	// === OPERATOR INTERFACE VALIDATION ===
	// Verify flags provide clear indication to operators
	IF eTestResult = E_CommandResult.Ok THEN
		AssertTrue(
			Condition := (iTestCommand.P_CommandStatus.BaseStatus.Done = TRUE) AND
						 (iTestCommand.P_CommandStatus.BaseStatus.Busy = FALSE) AND
						 (iTestCommand.P_CommandStatus.BaseStatus.Error = FALSE),
			Message := CONCAT(sTestScenario, ': OPERATOR - Success indication: Done=TRUE + Busy=FALSE + Error=FALSE')
		);
	ELSE
		AssertTrue(
			Condition := (iTestCommand.P_CommandStatus.BaseStatus.Error = TRUE) AND
						 (iTestCommand.P_CommandStatus.BaseStatus.Busy = FALSE),
			Message := CONCAT(sTestScenario, ': OPERATOR - Error indication: Error=TRUE + Busy=FALSE')
		);
	END_IF

	// Reset for next iteration
	iTestCommand.Reset();
END_FOR

TEST_FINISHED();
END_METHOD

METHOD PRIVATE TEST_Config_FallbackToLocal_WhenInjectedInvalid
VAR
	TestIdx : DINT := INDEX_CONFIG_FALLBACKTOLOCAL_WHENINJECTEDINVALID;
    configResolution : E_ConfigurationResolution;
END_VAR
TEST(__POUNAME());

// Purpose: Verify command falls back to local configuration when injected interfaces become invalid
// Tests resilient configuration resolution

// Initialize test objects - Use index 204 to avoid conflicts
TestCommand[TestIdx].Initialize();
TestComponent[TestIdx].Initialize();
TestCommandConfig[TestIdx].Initialize();
TestPermIntlk[TestIdx].Initialize();

// Safe interface assignments using __QUERYINTERFACE for validation
iTestCommand := TestCommand[TestIdx];

iTestCommandConfig := TestCommandConfig[TestIdx];

iTestComponent := TestComponent[TestIdx];

iTestPermIntlkConfig := TestPermIntlk[TestIdx];

// Interface validation
IF iTestCommand = 0 THEN
    AssertTrue(Condition := FALSE, Message := 'TEST FAILED: iTestCommand interface is null');
    RETURN;
END_IF

// === STEP 1: Initially Use Local Configuration ===
// Don't inject configurations - should use local fallback
TestCommand[TestIdx].Initialize();

// Verify local configuration is being used
configResolution := TestCommand[TestIdx].P_CommandStatus.CmdConfigurationResolution;
AssertEquals_INT(
    Expected := E_ConfigurationResolution.Local,
    Actual := configResolution,
    Message := 'Should use Local configuration when no interfaces injected'
);

// === STEP 2: Inject Valid Configurations ===
// Configure valid injected configuration
TestCommandConfig[TestIdx].P_CommandConfiguration.CommandDescription := 'Injected Valid Config';
TestCommandConfig[TestIdx].P_CommandConfiguration.TimeoutTime := T#15S;
TestCommandConfig[TestIdx].P_CommandConfiguration.RetryCountONLYFORCOMMSENDS := 5;

// Configure permissive to be OK for successful validation and execution
IF iTestPermIntlkConfig <> 0 THEN
	iTestPermIntlkConfig.P_PermIntlkConfiguration.PermIntlkObj[1].Description := 'Fallback Test Permissive';
	iTestPermIntlkConfig.P_PermIntlkConfiguration.PermIntlkObj[1].Condition := TRUE;
	iTestPermIntlkConfig.P_PermIntlkConfiguration.PermIntlkObj[1].Index := 1;
	TestPermIntlk[TestIdx].CyclicLogic(); // Update permissive evaluation
END_IF

// Inject configurations
iTestCommand.InjectConfigurations(
    iComponent := iTestComponent,
    iCommandConfiguration := iTestCommandConfig,
    iPermIntlkConfiguration := iTestPermIntlkConfig
);

// Resolve configurations after injection
iTestCommand.CyclicLogic();

// Verify injected configuration is being used
configResolution := iTestCommand.P_CommandStatus.CmdConfigurationResolution;
AssertEquals_INT(
    Expected := E_ConfigurationResolution.InjectedInterface,
    Actual := configResolution,
    Message := 'Should use InjectedInterface configuration when valid interfaces provided'
);

// Verify we can access injected configuration
AssertEquals_STRING(
    Expected := 'Injected Valid Config',
    Actual := TestCommand[TestIdx].P_CommandStatus.ConfigRef.CommandDescription,
    Message := 'Should access injected configuration description'
);

AssertEquals_TIME(
    Expected := T#15S,
    Actual := TestCommand[TestIdx].P_CommandStatus.ConfigRef.TimeoutTime,
    Message := 'Should access injected configuration timeout'
);

// === STEP 3: Simulate Configuration Becoming Invalid ===
// This tests runtime resilience when external configuration becomes corrupted
// In real systems, this could happen due to network issues, memory corruption, etc.

// Inject null interfaces to simulate failure
iTestCommand.InjectConfigurations(
    iComponent := iTestComponent,
    iCommandConfiguration := 0, // Null interface
    iPermIntlkConfiguration := 0  // Null interface
);

// Re-initialize to trigger configuration resolution
TestCommand[TestIdx].Initialize();

// Trigger configuration resolution after invalidation
iTestCommand.CyclicLogic();

// === STEP 4: Verify Fallback to Local Configuration ===
configResolution := TestCommand[TestIdx].P_CommandStatus.CmdConfigurationResolution;
AssertEquals_INT(
    Expected := E_ConfigurationResolution.Local,
    Actual := configResolution,
    Message := 'RESILIENCE: Should fallback to Local configuration when injected becomes invalid'
);

// Verify local configuration is accessible and provides default values
AssertEquals_STRING(
    Expected := 'Missing Command Configuration Interface Reference',
    Actual := TestCommand[TestIdx].LocalCommandConfiguration.CommandDescription,
    Message := 'Should use local fallback configuration description'
);

// === STEP 5: Command Should Still Function with Local Configuration ===
// Even with fallback configuration, basic command operations should work
iTestCommand.Execute();

// Command should accept execution even with local configuration
AssertEquals_UDINT(
    Expected := E_CommandResult.Accepted,
    Actual := iTestCommand.P_CommandStatus.Result,
    Message := 'Command should function with local fallback configuration'
);

// Progress through states
iTestCommand.CyclicLogic(); // Idle → Execute
iTestCommand.CyclicLogic(); // Execute → Monitor
iTestCommand.Complete(); // Signal completion
iTestCommand.CyclicLogic(); // Monitor → Complete

// Should complete successfully
AssertEquals_UDINT(
    Expected := E_CommandState.Complete,
    Actual := iTestCommand.P_CommandStatus.StepState,
    Message := 'Command should complete successfully with local configuration'
);

AssertEquals_UDINT(
    Expected := E_CommandResult.Ok,
    Actual := iTestCommand.P_CommandStatus.Result,
    Message := 'Command should have Ok result with local configuration'
);

TEST_FINISHED();
END_METHOD

METHOD PRIVATE TEST_Config_RecoveryToInjected_WhenValidAgain
VAR
	TestIdx : DINT := INDEX_CONFIG_RECOVERYTOINJECTED_WHENVALIDAGAIN;
    configResolution : E_ConfigurationResolution;
END_VAR
TEST(__POUNAME());

// Purpose: Verify command can recover to injected configuration when it becomes valid again
// Tests configuration resolution recovery mechanism

// Initialize test objects - Use index 205 to avoid conflicts
TestCommand[TestIdx].Initialize();
TestComponent[TestIdx].Initialize();
TestCommandConfig[TestIdx].Initialize();
TestPermIntlk[TestIdx].Initialize();

// Safe interface assignments using __QUERYINTERFACE for validation
iTestCommand := TestCommand[TestIdx];

iTestCommandConfig := TestCommandConfig[TestIdx];

iTestComponent := TestComponent[TestIdx];

iTestPermIntlkConfig := TestPermIntlk[TestIdx];

// Interface validation
IF iTestCommand = 0 THEN
    AssertTrue(Condition := FALSE, Message := 'TEST FAILED: iTestCommand interface is null');
    RETURN;
END_IF

// === STEP 1: Start with Local Configuration ===
TestCommand[TestIdx].Initialize();

configResolution := TestCommand[TestIdx].P_CommandStatus.CmdConfigurationResolution;
AssertEquals_INT(
    Expected := E_ConfigurationResolution.Local,
    Actual := configResolution,
    Message := 'Should start with Local configuration'
);

// === STEP 2: Inject Invalid Configuration (Null Interfaces) ===
iTestCommand.InjectConfigurations(
    iComponent := iTestComponent,
    iCommandConfiguration := 0, // Null interface
    iPermIntlkConfiguration := 0  // Null interface
);

TestCommand[TestIdx].Initialize();

// Should still use local configuration
configResolution := TestCommand[TestIdx].P_CommandStatus.CmdConfigurationResolution;
AssertEquals_INT(
    Expected := E_ConfigurationResolution.Local,
    Actual := configResolution,
    Message := 'Should remain with Local configuration when invalid injected'
);

// === STEP 3: Inject Valid Configuration ===
// Configure a distinctive injected configuration for recovery test
TestCommandConfig[TestIdx].P_CommandConfiguration.CommandDescription := 'Recovered Injected Config';
TestCommandConfig[TestIdx].P_CommandConfiguration.TimeoutTime := T#25S;
TestCommandConfig[TestIdx].P_CommandConfiguration.RetryCountONLYFORCOMMSENDS := 7;

// Configure permissive to be OK for successful validation and execution
IF iTestPermIntlkConfig <> 0 THEN
	iTestPermIntlkConfig.P_PermIntlkConfiguration.PermIntlkObj[1].Description := 'Recovery Test Permissive';
	iTestPermIntlkConfig.P_PermIntlkConfiguration.PermIntlkObj[1].Condition := TRUE;
	iTestPermIntlkConfig.P_PermIntlkConfiguration.PermIntlkObj[1].Index := 1;
	TestPermIntlk[TestIdx].CyclicLogic(); // Update permissive evaluation
END_IF

// Inject valid configurations
iTestCommand.InjectConfigurations(
    iComponent := iTestComponent,
    iCommandConfiguration := iTestCommandConfig,
    iPermIntlkConfiguration := iTestPermIntlkConfig
);

// Resolve configurations after injection
iTestCommand.CyclicLogic();

// Re-initialize to trigger configuration resolution
TestCommand[TestIdx].Initialize();

// === STEP 4: Verify Recovery to Injected Configuration ===
configResolution := TestCommand[TestIdx].P_CommandStatus.CmdConfigurationResolution;
AssertEquals_INT(
    Expected := E_ConfigurationResolution.InjectedInterface,
    Actual := configResolution,
    Message := 'RECOVERY: Should recover to InjectedInterface when valid again'
);

// Verify recovered configuration is accessible
AssertEquals_STRING(
    Expected := 'Recovered Injected Config',
    Actual := TestCommand[TestIdx].P_CommandStatus.ConfigRef.CommandDescription,
    Message := 'Should access recovered injected configuration description'
);

AssertEquals_TIME(
    Expected := T#25S,
    Actual := TestCommand[TestIdx].P_CommandStatus.ConfigRef.TimeoutTime,
    Message := 'Should access recovered injected configuration timeout'
);

AssertEquals_DINT(
    Expected := 7,
    Actual := TestCommand[TestIdx].P_CommandStatus.ConfigRef.RetryCountONLYFORCOMMSENDS,
    Message := 'Should access recovered injected configuration retry count'
);

// === STEP 5: Command Should Function with Recovered Configuration ===
iTestCommand.Execute();

AssertEquals_UDINT(
    Expected := E_CommandResult.Accepted,
    Actual := iTestCommand.P_CommandStatus.Result,
    Message := 'Command should function with recovered configuration'
);

// Progress through states with recovered configuration
iTestCommand.CyclicLogic(); // Idle → Execute
iTestCommand.CyclicLogic(); // Execute → Monitor
iTestCommand.Complete(); // Signal completion
iTestCommand.CyclicLogic(); // Monitor → Complete

AssertEquals_UDINT(
    Expected := E_CommandState.Complete,
    Actual := iTestCommand.P_CommandStatus.StepState,
    Message := 'Command should complete with recovered configuration'
);

AssertEquals_UDINT(
    Expected := E_CommandResult.Ok,
    Actual := iTestCommand.P_CommandStatus.Result,
    Message := 'Command should have Ok result with recovered configuration'
);

// === STEP 6: Test Multiple Recovery Cycles ===
// Simulate configuration becoming invalid again, then valid
iTestCommand.InjectConfigurations(
    iComponent := iTestComponent,
    iCommandConfiguration := 0, // Invalid again
    iPermIntlkConfiguration := 0
);

TestCommand[TestIdx].Initialize();

configResolution := TestCommand[TestIdx].P_CommandStatus.CmdConfigurationResolution;
AssertEquals_INT(
    Expected := E_ConfigurationResolution.Local,
    Actual := configResolution,
    Message := 'Should fallback to Local when invalid again'
);

// Recover again
TestCommandConfig[TestIdx].P_CommandConfiguration.CommandDescription := 'Second Recovery Config';
iTestCommand.InjectConfigurations(
    iComponent := iTestComponent,
    iCommandConfiguration := iTestCommandConfig,
    iPermIntlkConfiguration := iTestPermIntlkConfig
);

// Resolve configurations after second injection
iTestCommand.CyclicLogic();

TestCommand[TestIdx].Initialize();

configResolution := TestCommand[TestIdx].P_CommandStatus.CmdConfigurationResolution;
AssertEquals_INT(
    Expected := E_ConfigurationResolution.InjectedInterface,
    Actual := configResolution,
    Message := 'RESILIENCE: Should recover multiple times'
);

AssertEquals_STRING(
    Expected := 'Second Recovery Config',
    Actual := TestCommand[TestIdx].P_CommandStatus.ConfigRef.CommandDescription,
    Message := 'Should access second recovery configuration'
);

TEST_FINISHED();
END_METHOD

METHOD PRIVATE TEST_Execute_ValidatesBeforeAccepting
VAR
	TestIdx : DINT := INDEX_EXECUTE_VALIDATESBEFOREACCEPTING;
	stCommandStatus : ST_CommandStatus;
	stBaseStatus : ST_BaseStatus;
	stCommandConfiguration : ST_CommandConfiguration;
	ValidationCallCount : INT := 0;
	i : DINT;
END_VAR
TEST(__POUNAME());
// Purpose: Guards that Execute always re-validates before setting Accepted.
// Impact: Prevents stale validation results from allowing unsafe execution.
// Reference: FB_Command.TcPOU Execute() method and validation integration

// Initialize reference objects for stCommandStatus
stCommandStatus.BaseStatus REF= stBaseStatus;
stCommandStatus.ConfigRef REF= stCommandConfiguration;

// === TEST SCENARIO 1: Execute() with Valid Conditions ===
// Initialize test objects first - Use index 121 to avoid conflicts
TestCommand[TestIdx].Initialize();
TestComponent[TestIdx].Initialize();
TestCommandConfig[TestIdx].Initialize();
TestPermIntlk[TestIdx].Initialize();

// Safe interface assignments using __QUERYINTERFACE for validation
iTestCommand := TestCommand[TestIdx];

iTestCommandConfig := TestCommandConfig[TestIdx];

iTestComponent := TestComponent[TestIdx];

iTestPermIntlkConfig := TestPermIntlk[TestIdx];

// Configure command for validation testing
TestCommandConfig[TestIdx].P_CommandConfiguration.CommandDescription := 'Execute Validation Test - Valid Conditions';
IF __ISVALIDREF(TestCommandConfig[TestIdx].P_CommandConfiguration.BaseConfiguration) THEN
    TestCommandConfig[TestIdx].P_CommandConfiguration.BaseConfiguration.LogTraceConfiguration.When := E_LogTraceWhen.xRunOnInitOnly;
END_IF
TestCommandConfig[TestIdx].P_CommandConfiguration.TimeoutTime := T#30S;
TestCommandConfig[TestIdx].P_CommandConfiguration.PermIntlkConfiguredAsInterlock := TRUE;

// Setup valid permissives
IF iTestPermIntlkConfig <> 0 THEN
	iTestPermIntlkConfig.P_PermIntlkConfiguration.PermIntlkObj[1].Description := 'Execute Validation Test Permissive';
	iTestPermIntlkConfig.P_PermIntlkConfiguration.PermIntlkObj[1].Condition := TRUE;
	iTestPermIntlkConfig.P_PermIntlkConfiguration.PermIntlkObj[1].Index := 1;
	TestPermIntlk[TestIdx].CyclicLogic(); // Update permissive evaluation
END_IF

// Setup command with configurations
iTestCommand.InjectConfigurations(
	iComponent := iTestComponent,
	iCommandConfiguration := iTestCommandConfig,
	iPermIntlkConfiguration := iTestPermIntlkConfig
);

// Verify initial state
AssertEquals_UDINT(
	Expected := E_CommandState.Idle,
	Actual := iTestCommand.P_CommandStatus.StepState,
	Message := 'VALIDATION TEST: Command should start in Idle state'
);

AssertEquals_UDINT(
	Expected := E_CommandResult.None,
	Actual := iTestCommand.P_CommandStatus.Result,
	Message := 'VALIDATION TEST: Command should start with None result'
);

// === CRITICAL TEST: Execute() Should Re-Validate Before Accepting ===
// This is the core test - Execute() must not rely on stale validation results
iTestCommand.Execute();

// Verify Execute() performed validation and accepted based on current conditions
AssertEquals_UDINT(
	Expected := E_CommandResult.Accepted,
	Actual := iTestCommand.P_CommandStatus.Result,
	Message := 'EXECUTE VALIDATION: Execute() must validate and accept when conditions are valid'
);

AssertTrue(
	Condition := iTestCommand.P_CommandStatus.BaseStatus.Busy,
	Message := 'EXECUTE VALIDATION: Accepted command should set Busy=TRUE'
);

// === TEST SCENARIO 2: Execute() with Invalid Conditions ===
// Reset and test with invalid conditions
TestCommand[TestIdx].Initialize();
TestComponent[TestIdx].Initialize();
TestCommandConfig[TestIdx].Initialize();
TestPermIntlk[TestIdx].Initialize();

// Safe interface assignments
iTestCommand := TestCommand[TestIdx];

iTestCommandConfig := TestCommandConfig[TestIdx];

iTestComponent := TestComponent[TestIdx];

iTestPermIntlkConfig := TestPermIntlk[TestIdx];

// Configure command for failed validation test
TestCommandConfig[TestIdx].P_CommandConfiguration.CommandDescription := 'Execute Validation Test - Invalid Conditions';
IF __ISVALIDREF(TestCommandConfig[TestIdx].P_CommandConfiguration.BaseConfiguration) THEN
    TestCommandConfig[TestIdx].P_CommandConfiguration.BaseConfiguration.LogTraceConfiguration.When := E_LogTraceWhen.xRunOnInitOnly;
END_IF
TestCommandConfig[TestIdx].P_CommandConfiguration.TimeoutTime := T#30S;
TestCommandConfig[TestIdx].P_CommandConfiguration.PermIntlkConfiguredAsInterlock := TRUE;

// Setup INVALID permissives - this should cause validation failure
IF iTestPermIntlkConfig <> 0 THEN
	iTestPermIntlkConfig.P_PermIntlkConfiguration.PermIntlkObj[1].Description := 'Execute Validation Test Failed Permissive';
	iTestPermIntlkConfig.P_PermIntlkConfiguration.PermIntlkObj[1].Condition := FALSE; // INVALID!
	iTestPermIntlkConfig.P_PermIntlkConfiguration.PermIntlkObj[1].Index := 1;
	TestPermIntlk[TestIdx].CyclicLogic(); // Update permissive evaluation
END_IF

// Setup command with configurations
iTestCommand.InjectConfigurations(
	iComponent := iTestComponent,
	iCommandConfiguration := iTestCommandConfig,
	iPermIntlkConfiguration := iTestPermIntlkConfig
);

// === CRITICAL TEST: Execute() Should Reject When Validation Fails ===
// Execute() must validate current conditions and reject if invalid
iTestCommand.Execute();

// Verify Execute() detected invalid conditions and rejected execution
AssertEquals_UDINT(
	Expected := E_CommandResult.Forbidden,
	Actual := iTestCommand.P_CommandStatus.Result,
	Message := 'EXECUTE VALIDATION: Execute() must validate and reject when conditions are invalid'
);

AssertFalse(
	Condition := iTestCommand.P_CommandStatus.BaseStatus.Busy,
	Message := 'EXECUTE VALIDATION: Rejected command should keep Busy=FALSE'
);

AssertTrue(
	Condition := iTestCommand.P_CommandStatus.BaseStatus.Error,
	Message := 'EXECUTE VALIDATION: Forbidden result should set Error=TRUE'
);

// === TEST SCENARIO 3: Stale Validation Prevention ===
// Test that Execute() doesn't rely on previous validation results
TestCommand[TestIdx].Initialize();
TestComponent[TestIdx].Initialize();
TestCommandConfig[TestIdx].Initialize();
TestPermIntlk[TestIdx].Initialize();

// Safe interface assignments
iTestCommand := TestCommand[TestIdx];

iTestCommandConfig := TestCommandConfig[TestIdx];

iTestComponent := TestComponent[TestIdx];

iTestPermIntlkConfig := TestPermIntlk[TestIdx];

// Configure command for stale validation test
TestCommandConfig[TestIdx].P_CommandConfiguration.CommandDescription := 'Execute Validation Test - Stale Validation Prevention';
IF __ISVALIDREF(TestCommandConfig[TestIdx].P_CommandConfiguration.BaseConfiguration) THEN
    TestCommandConfig[TestIdx].P_CommandConfiguration.BaseConfiguration.LogTraceConfiguration.When := E_LogTraceWhen.xRunOnInitOnly;
END_IF
TestCommandConfig[TestIdx].P_CommandConfiguration.PermIntlkConfiguredAsInterlock := TRUE;

// Setup permissives initially valid
IF iTestPermIntlkConfig <> 0 THEN
	iTestPermIntlkConfig.P_PermIntlkConfiguration.PermIntlkObj[1].Description := 'Stale Validation Test Permissive';
	iTestPermIntlkConfig.P_PermIntlkConfiguration.PermIntlkObj[1].Condition := TRUE;
	iTestPermIntlkConfig.P_PermIntlkConfiguration.PermIntlkObj[1].Index := 1;
	TestPermIntlk[TestIdx].CyclicLogic(); // Update permissive evaluation
END_IF

// Setup command with configurations
iTestCommand.InjectConfigurations(
	iComponent := iTestComponent,
	iCommandConfiguration := iTestCommandConfig,
	iPermIntlkConfiguration := iTestPermIntlkConfig
);

// Perform initial validation (this would be successful)
iTestCommand.Validate();

AssertEquals_UDINT(
	Expected := E_CommandResult.Accepted,
	Actual := iTestCommand.P_CommandStatus.Result,
	Message := 'STALE VALIDATION: Initial validation should succeed'
);

// === CRITICAL: Change Conditions After Validation ===
// This simulates the stale validation scenario
IF iTestPermIntlkConfig <> 0 THEN
	iTestPermIntlkConfig.P_PermIntlkConfiguration.PermIntlkObj[1].Condition := FALSE; // Make invalid!
	TestPermIntlk[TestIdx].CyclicLogic(); // Update permissive evaluation
END_IF

// === CRITICAL TEST: Execute() Must Re-Validate (Not Use Stale Result) ===
// Execute() should detect the changed conditions and reject, despite previous successful validation
iTestCommand.Execute();

// Verify Execute() performed fresh validation and detected the changed conditions
AssertEquals_UDINT(
	Expected := E_CommandResult.Forbidden,
	Actual := iTestCommand.P_CommandStatus.Result,
	Message := 'STALE VALIDATION PREVENTION: Execute() must re-validate and detect changed conditions'
);

AssertFalse(
	Condition := iTestCommand.P_CommandStatus.BaseStatus.Busy,
	Message := 'STALE VALIDATION PREVENTION: Command should not start with invalid conditions'
);

AssertTrue(
	Condition := iTestCommand.P_CommandStatus.BaseStatus.Error,
	Message := 'STALE VALIDATION PREVENTION: Changed conditions should result in Error=TRUE'
);

// === TEST SCENARIO 4: Validation-Execute Integration ===
// Test the complete validation-execute flow
TestCommand[TestIdx].Initialize();
TestComponent[TestIdx].Initialize();
TestCommandConfig[TestIdx].Initialize();
TestPermIntlk[TestIdx].Initialize();

// Safe interface assignments
iTestCommand := TestCommand[TestIdx];

iTestCommandConfig := TestCommandConfig[TestIdx];

iTestComponent := TestComponent[TestIdx];

iTestPermIntlkConfig := TestPermIntlk[TestIdx];

// Configure command for integration test
TestCommandConfig[TestIdx].P_CommandConfiguration.CommandDescription := 'Execute Validation Test - Integration';
IF __ISVALIDREF(TestCommandConfig[TestIdx].P_CommandConfiguration.BaseConfiguration) THEN
    TestCommandConfig[TestIdx].P_CommandConfiguration.BaseConfiguration.LogTraceConfiguration.When := E_LogTraceWhen.xRunOnInitOnly;
END_IF
TestCommandConfig[TestIdx].P_CommandConfiguration.PermIntlkConfiguredAsInterlock := TRUE;

// Setup valid permissives
IF iTestPermIntlkConfig <> 0 THEN
	iTestPermIntlkConfig.P_PermIntlkConfiguration.PermIntlkObj[1].Description := 'Integration Test Permissive';
	iTestPermIntlkConfig.P_PermIntlkConfiguration.PermIntlkObj[1].Condition := TRUE;
	iTestPermIntlkConfig.P_PermIntlkConfiguration.PermIntlkObj[1].Index := 1;
	TestPermIntlk[TestIdx].CyclicLogic(); // Update permissive evaluation
END_IF

// Setup command with configurations
iTestCommand.InjectConfigurations(
	iComponent := iTestComponent,
	iCommandConfiguration := iTestCommandConfig,
	iPermIntlkConfiguration := iTestPermIntlkConfig
);

// Call Validate() explicitly first
iTestCommand.Validate();

AssertEquals_UDINT(
	Expected := E_CommandResult.Accepted,
	Actual := iTestCommand.P_CommandStatus.Result,
	Message := 'INTEGRATION: Explicit validation should succeed'
);

// Now call Execute() - should still re-validate and accept
iTestCommand.Execute();

AssertEquals_UDINT(
	Expected := E_CommandResult.Accepted,
	Actual := iTestCommand.P_CommandStatus.Result,
	Message := 'INTEGRATION: Execute() should re-validate and accept consistent conditions'
);

AssertTrue(
	Condition := iTestCommand.P_CommandStatus.BaseStatus.Busy,
	Message := 'INTEGRATION: Successfully validated and executed command should be Busy'
);

// Verify command starts executing
iTestCommand.CyclicLogic();

AssertTrue(
	Condition := (iTestCommand.P_CommandStatus.StepState = E_CommandState.Execute) OR
				 (iTestCommand.P_CommandStatus.StepState = E_CommandState.Monitor),
	Message := 'INTEGRATION: Command should progress to Execute or Monitor state'
);

// === CLEANUP ===
// Reset all test commands
iTestCommand.Reset();

TEST_FINISHED();
END_METHOD

METHOD PRIVATE TEST_RuntimeCommandConfigLoss_InjectedRefsInvalidatedDuringExecution
VAR
	TestIdx : DINT := INDEX_RUNTIMECOMMANDCONFIGLOSS_INJECTEDREFSINVALIDATED;
    cmdResolution : E_ConfigurationResolution;
    permResolution : E_ConfigurationResolution;
    resultOK : E_CommandResult;
    commandDesc : STRING;
END_VAR
TEST(__POUNAME());

// Purpose: Test actual runtime configuration loss scenario where injected command/permintlk references
// become invalid during execution without explicit re-injection
// This validates our _EvaluateConfiguration fix that detects resolution changes for FB_Command

// === STEP 1: Set up valid injected configurations ===
TestCommand[TestIdx].Initialize();
TestComponent[TestIdx].Initialize();
TestCommandConfig[TestIdx].Initialize();
TestPermIntlk[TestIdx].Initialize();

// Configure distinctive injected configurations
TestCommandConfig[TestIdx].P_CommandConfiguration.CommandDescription := 'Runtime Valid Command Config';
TestCommandConfig[TestIdx].P_CommandConfiguration.TimeoutTime := T#30S;
TestCommandConfig[TestIdx].P_CommandConfiguration.RetryCountONLYFORCOMMSENDS := 3;

TestPermIntlk[TestIdx].P_PermIntlkConfiguration.Mode := E_ModePermIntlk.IfAllConditionsMet;
TestPermIntlk[TestIdx].P_PermIntlkConfiguration.PermIntlkObj[0].Description := 'Runtime Valid PermIntlk';
TestPermIntlk[TestIdx].P_PermIntlkConfiguration.PermIntlkObj[0].Condition := TRUE;

// Safe interface assignments
iTestCommand := TestCommand[TestIdx];
iTestCommandConfig := TestCommandConfig[TestIdx];
iTestComponent := TestComponent[TestIdx];
iTestPermIntlkConfig := TestPermIntlk[TestIdx];

// Inject configurations normally
iTestCommand.InjectConfigurations(
    iComponent := iTestComponent,
    iCommandConfiguration := iTestCommandConfig,
    iPermIntlkConfiguration := iTestPermIntlkConfig
);

// Resolve configurations after injection
iTestCommand.CyclicLogic();

// === STEP 2: Verify initially using injected configurations ===
cmdResolution := iTestCommand.P_CommandStatus.CmdConfigurationResolution;
permResolution := iTestCommand.P_CommandStatus.PermIntlkConfigResolution;

AssertEquals_DINT(Expected := TO_DINT(E_ConfigurationResolution.InjectedInterface), Actual := TO_DINT(cmdResolution), Message := 'Should initially use injected command configuration');
AssertEquals_DINT(Expected := TO_DINT(E_ConfigurationResolution.InjectedInterface), Actual := TO_DINT(permResolution), Message := 'Should initially use injected permintlk configuration');

// === STEP 3: Local fallback configurations will use defaults ===

// === STEP 4: Simulate runtime reference invalidation ===
// This simulates what happens when network connections are lost, memory corruption occurs,
// or external systems become unavailable - WITHOUT calling InjectConfigurations again
// We simulate this by calling InjectConfigurations with null interfaces to trigger the runtime scenario
iTestCommand.InjectConfigurations(
    iComponent := iTestComponent,
    iCommandConfiguration := 0,        // Simulate command config becoming invalid
    iPermIntlkConfiguration := 0       // Simulate permintlk config becoming invalid
);

// === STEP 5: Trigger resolution change detection through CyclicLogic ===
// Our fix should detect the resolution changes and update references
iTestCommand.CyclicLogic();

// === STEP 6: Verify automatic fallback to local configurations ===
cmdResolution := TestCommand[TestIdx].P_CommandStatus.CmdConfigurationResolution;
permResolution := TestCommand[TestIdx].P_CommandStatus.PermIntlkConfigResolution;
commandDesc := TestCommand[TestIdx].P_CommandStatus.ConfigRef.CommandDescription;

AssertEquals_DINT(Expected := TO_DINT(E_ConfigurationResolution.Local), Actual := TO_DINT(cmdResolution), Message := 'RUNTIME FIX: Should automatically switch to local command configuration when injected refs become invalid');
AssertEquals_DINT(Expected := TO_DINT(E_ConfigurationResolution.Local), Actual := TO_DINT(permResolution), Message := 'RUNTIME FIX: Should automatically switch to local permintlk configuration when injected refs become invalid');
AssertEquals_STRING(Expected := 'Missing Command Configuration Interface Reference', Actual := commandDesc, Message := 'Should use local fallback command configuration description');

// === STEP 7: Verify continued command operation with local configuration ===
// Command should still function with local fallback configuration
iTestCommand.Execute();
resultOK := iTestCommand.P_CommandStatus.Result;

AssertEquals_UDINT(Expected := E_CommandResult.Accepted, Actual := resultOK, Message := 'Command should accept execution with local fallback configuration');

// Progress through command states
iTestCommand.CyclicLogic(); // Idle → Execute
iTestCommand.CyclicLogic(); // Execute → Monitor
iTestCommand.CyclicLogic(); // Monitor → Complete

AssertEquals_UDINT(Expected := E_CommandState.Complete, Actual := iTestCommand.P_CommandStatus.StepState, Message := 'Command should complete successfully with local configuration');
AssertEquals_UDINT(Expected := E_CommandResult.Ok, Actual := iTestCommand.P_CommandStatus.Result, Message := 'Command should have Ok result with local configuration');

// === STEP 8: Verify stable operation over multiple cycles ===
iTestCommand.CyclicLogic(); // Auto-reset cycle
iTestCommand.CyclicLogic(); // Additional stability check

cmdResolution := TestCommand[TestIdx].P_CommandStatus.CmdConfigurationResolution;
permResolution := TestCommand[TestIdx].P_CommandStatus.PermIntlkConfigResolution;

AssertEquals_DINT(Expected := TO_DINT(E_ConfigurationResolution.Local), Actual := TO_DINT(cmdResolution), Message := 'Should maintain local command configuration resolution consistently');
AssertEquals_DINT(Expected := TO_DINT(E_ConfigurationResolution.Local), Actual := TO_DINT(permResolution), Message := 'Should maintain local permintlk configuration resolution consistently');

TEST_FINISHED();
END_METHOD

METHOD PRIVATE TEST_RuntimeCommandConfigRecovery_ValidRefsRestoredDuringExecution
VAR
	TestIdx : DINT := INDEX_RUNTIMECOMMANDCONFIGRECOVERY_VALIDREFSRESTORED;
    cmdResolution : E_ConfigurationResolution;
    permResolution : E_ConfigurationResolution;
    resultOK : E_CommandResult;
    commandDesc : STRING;
    timeoutTime : TIME;
END_VAR
TEST(__POUNAME());

// Purpose: Test runtime configuration recovery scenario where injected command/permintlk references
// are restored during execution after being invalid
// This validates our _EvaluateConfiguration fix for bidirectional resolution changes for FB_Command

// === STEP 1: Start with local configurations ===
TestCommand[TestIdx].Initialize();
TestComponent[TestIdx].Initialize();
TestCommandConfig[TestIdx].Initialize();
TestPermIntlk[TestIdx].Initialize();

// Safe interface assignment for command only
iTestCommand := TestCommand[TestIdx];

TestCommand[TestIdx].CyclicLogic();

// Verify starting with local configurations
cmdResolution := TestCommand[TestIdx].P_CommandStatus.CmdConfigurationResolution;
permResolution := TestCommand[TestIdx].P_CommandStatus.PermIntlkConfigResolution;

AssertEquals_DINT(Expected := TO_DINT(E_ConfigurationResolution.Local), Actual := TO_DINT(cmdResolution), Message := 'Should start with local command configuration');
AssertEquals_DINT(Expected := TO_DINT(E_ConfigurationResolution.Local), Actual := TO_DINT(permResolution), Message := 'Should start with local permintlk configuration');

// === STEP 2: Set up distinctive injected configurations ===
TestCommandConfig[TestIdx].P_CommandConfiguration.CommandDescription := 'Recovery Injected Command Config';
TestCommandConfig[TestIdx].P_CommandConfiguration.TimeoutTime := T#45S;
TestCommandConfig[TestIdx].P_CommandConfiguration.RetryCountONLYFORCOMMSENDS := 8;

TestPermIntlk[TestIdx].P_PermIntlkConfiguration.Mode := E_ModePermIntlk.IfAllConditionsMet;
TestPermIntlk[TestIdx].P_PermIntlkConfiguration.PermIntlkObj[1].Description := 'Recovery Injected PermIntlk';
TestPermIntlk[TestIdx].P_PermIntlkConfiguration.PermIntlkObj[1].Condition := TRUE;
TestPermIntlk[TestIdx].P_PermIntlkConfiguration.PermIntlkObj[1].Index := 1;

// Safe interface assignments for injected configurations
iTestCommandConfig := TestCommandConfig[TestIdx];
iTestComponent := TestComponent[TestIdx];
iTestPermIntlkConfig := TestPermIntlk[TestIdx];

// === STEP 3: Simulate runtime reference restoration ===
// This simulates what happens when network connections are restored, external systems
// come back online, or memory references are re-established - WITHOUT calling InjectConfigurations again
// We restore the interface references to simulate runtime recovery
iTestCommand.InjectConfigurations(
    iComponent := iTestComponent,
    iCommandConfiguration := iTestCommandConfig,        // Simulate command config becoming valid again
    iPermIntlkConfiguration := iTestPermIntlkConfig     // Simulate permintlk config becoming valid again
);

// === STEP 4: Trigger resolution change detection through CyclicLogic ===
// Our fix should detect the resolution changes and update references
iTestCommand.CyclicLogic();

// === STEP 5: Verify automatic recovery to injected configurations ===
cmdResolution := TestCommand[TestIdx].P_CommandStatus.CmdConfigurationResolution;
permResolution := TestCommand[TestIdx].P_CommandStatus.PermIntlkConfigResolution;
commandDesc := TestCommand[TestIdx].P_CommandStatus.ConfigRef.CommandDescription;
timeoutTime := TestCommand[TestIdx].P_CommandStatus.ConfigRef.TimeoutTime;

AssertEquals_DINT(Expected := TO_DINT(E_ConfigurationResolution.InjectedInterface), Actual := TO_DINT(cmdResolution), Message := 'RUNTIME FIX: Should automatically switch to injected command configuration when refs become valid');
AssertEquals_DINT(Expected := TO_DINT(E_ConfigurationResolution.InjectedInterface), Actual := TO_DINT(permResolution), Message := 'RUNTIME FIX: Should automatically switch to injected permintlk configuration when refs become valid');
AssertEquals_STRING(Expected := 'Recovery Injected Command Config', Actual := commandDesc, Message := 'Should use recovered injected command configuration description');
AssertEquals_TIME(Expected := T#45S, Actual := timeoutTime, Message := 'Should use recovered injected command configuration timeout');

// === STEP 6: Verify command functions correctly with recovered configuration ===
iTestCommand.Execute();
resultOK := iTestCommand.P_CommandStatus.Result;

AssertEquals_UDINT(Expected := E_CommandResult.Accepted, Actual := resultOK, Message := 'Command should accept execution with recovered injected configuration');

// Progress through command states with recovered configuration
iTestCommand.CyclicLogic(); // Idle → Execute
iTestCommand.CyclicLogic(); // Execute → Monitor
iTestCommand.CyclicLogic(); // Monitor → Complete

AssertEquals_UDINT(Expected := E_CommandState.Complete, Actual := iTestCommand.P_CommandStatus.StepState, Message := 'Command should complete successfully with recovered configuration');
AssertEquals_UDINT(Expected := E_CommandResult.Ok, Actual := iTestCommand.P_CommandStatus.Result, Message := 'Command should have Ok result with recovered configuration');

// === STEP 7: Verify stable operation over multiple cycles ===
iTestCommand.CyclicLogic(); // Auto-reset cycle
iTestCommand.CyclicLogic(); // Additional stability check

cmdResolution := TestCommand[TestIdx].P_CommandStatus.CmdConfigurationResolution;
permResolution := TestCommand[TestIdx].P_CommandStatus.PermIntlkConfigResolution;

AssertEquals_DINT(Expected := TO_DINT(E_ConfigurationResolution.InjectedInterface), Actual := TO_DINT(cmdResolution), Message := 'Should maintain injected command configuration resolution consistently');
AssertEquals_DINT(Expected := TO_DINT(E_ConfigurationResolution.InjectedInterface), Actual := TO_DINT(permResolution), Message := 'Should maintain injected permintlk configuration resolution consistently');

TEST_FINISHED();
END_METHOD

METHOD PRIVATE TEST_AbortDuringCompletionWait
VAR_INST
	AbortCycles : INT := 0;
	CompletionCondition	: BOOL;
END_VAR
VAR
	TestName : Tc2_System.T_MaxString := 'TEST_AbortDuringCompletionWait';
	TestIdx : DINT := INDEX_ABORTDURINGCOMPLETIONWAIT;
END_VAR
TEST(__POUNAME());

// Initialize test objects on first cycle only
IF AbortCycles = 0 THEN
	TestCommand[TestIdx].Initialize();
	TestComponent[TestIdx].Initialize();
	TestCommandConfig[TestIdx].Initialize();
	TestPermIntlk[TestIdx].Initialize();

	// Safe interface assignments
	iTestCommand := TestCommand[TestIdx];
	iTestCommandConfig := TestCommandConfig[TestIdx];
	iTestComponent := TestComponent[TestIdx];
	iTestPermIntlkConfig := TestPermIntlk[TestIdx];

	// Interface validation with protection
	IF iTestCommand = 0 THEN
		AssertTrue(Condition := FALSE, Message := 'TEST FAILED: iTestCommand interface is null');
		AbortCycles := 0;
		RETURN;
	END_IF

	IF iTestCommandConfig = 0 THEN
		AssertTrue(Condition := FALSE, Message := 'TEST FAILED: iTestCommandConfig interface is null');
		AbortCycles := 0;
		RETURN;
	END_IF

	IF iTestComponent = 0 THEN
		AssertTrue(Condition := FALSE, Message := 'TEST FAILED: iTestComponent interface is null');
		AbortCycles := 0;
		RETURN;
	END_IF

	// Configure command with completion condition that will take time (never reaches 10)
	CompletionCondition	:= (AbortCycles >= 10);
	iTestCommandConfig.P_CommandConfiguration.CompletionCondition REF= CompletionCondition; 
	iTestCommandConfig.P_CommandConfiguration.CommandDescription := 'Abort during completion wait test';
	iTestCommandConfig.P_CommandConfiguration.TimeoutTime := T#30S;
	IF __ISVALIDREF(iTestCommandConfig.P_CommandConfiguration.BaseConfiguration) THEN
		iTestCommandConfig.P_CommandConfiguration.BaseConfiguration.LogTraceConfiguration.When := E_LogTraceWhen.xRunOnInitOnly;
	END_IF

	// Setup component to be enabled and not busy
	IF iTestComponent <> 0 THEN
		iTestComponent.P_ComponentStatus.BaseStatus.Enabled := TRUE;
		iTestComponent.P_ComponentStatus.BaseStatus.Busy := FALSE;
		iTestComponent.P_ComponentStatus.BaseStatus.Error := FALSE;
	END_IF

	// Configure permissive to be OK
	IF iTestPermIntlkConfig <> 0 THEN
		iTestPermIntlkConfig.P_PermIntlkConfiguration.PermIntlkObj[1].Description := 'Abort Wait Permissive';
		iTestPermIntlkConfig.P_PermIntlkConfiguration.PermIntlkObj[1].Condition := TRUE;
		iTestPermIntlkConfig.P_PermIntlkConfiguration.PermIntlkObj[1].Index := 1;
		TestPermIntlk[TestIdx].CyclicLogic(); // Update permissive evaluation
	END_IF

	// Setup command with configurations
	iTestCommand.InjectConfigurations(
		iComponent := iTestComponent,
		iCommandConfiguration := iTestCommandConfig,
		iPermIntlkConfiguration := iTestPermIntlkConfig
	);

	// Resolve configurations after injection
	iTestCommand.CyclicLogic();

	// Execute command
	iTestCommand.Execute();

	// Verify Execute() accepted the command
	AssertEquals_UDINT(
		Expected := E_CommandResult.Accepted,
		Actual := iTestCommand.P_CommandStatus.Result,
		Message := 'Execute() should set Result to Accepted'
	);
ELSE
	// Refresh interface references for subsequent cycles
	iTestCommand := TestCommand[TestIdx];
	iTestCommandConfig := TestCommandConfig[TestIdx];
END_IF

AbortCycles := AbortCycles + 1;

// Update completion condition dynamically
CompletionCondition	:= (AbortCycles >= 10);
iTestCommandConfig.P_CommandConfiguration.CompletionCondition ref= CompletionCondition;

// Run cyclic logic
iTestCommand.CyclicLogic();

// Abort command after 5 cycles (before completion condition becomes TRUE)
IF AbortCycles = 5 THEN
	iTestCommand.Abort();
END_IF

// Verify abort occurred after giving system time to process
IF AbortCycles = 7 THEN
	AssertEquals_UDINT(
		Expected := E_CommandResult.Aborted,
		Actual := iTestCommand.P_CommandStatus.Result,
		Message := 'Command should have Result=Aborted when aborted during completion wait'
	);

	AssertFalse(
		Condition := iTestCommand.P_CommandStatus.BaseStatus.Busy,
		Message := 'Command should clear Busy=FALSE after abort'
	);

	AssertEquals_UDINT(
		Expected := E_CommandState.Complete,
		Actual := iTestCommand.P_CommandStatus.StepState,
		Message := 'Command should be in Complete state after abort'
	);

	TEST_FINISHED();
	AbortCycles := 0;
END_IF
END_METHOD

METHOD PRIVATE TEST_CompletionCallbackToSequencer
VAR_INST
	SequenceCycles : INT := 0;
	SimulatedSequenceStep : INT := 0;
	CompletionCondition	: BOOL;
END_VAR
VAR
	TestName : Tc2_System.T_MaxString := 'TEST_CompletionCallbackToSequencer';
	TestIdx : DINT := INDEX_COMPLETIONCALLBACKTOSEQUENCER;
END_VAR
TEST(__POUNAME());

// Initialize test objects on first cycle only
IF SequenceCycles = 0 THEN
	TestCommand[TestIdx].Initialize();
	TestComponent[TestIdx].Initialize();
	TestCommandConfig[TestIdx].Initialize();
	TestPermIntlk[TestIdx].Initialize();

	// Safe interface assignments
	iTestCommand := TestCommand[TestIdx];
	iTestCommandConfig := TestCommandConfig[TestIdx];
	iTestComponent := TestComponent[TestIdx];
	iTestPermIntlkConfig := TestPermIntlk[TestIdx];

	// Interface validation with protection
	IF iTestCommand = 0 THEN
		AssertTrue(Condition := FALSE, Message := 'TEST FAILED: iTestCommand interface is null');
		SequenceCycles := 0;
		RETURN;
	END_IF

	IF iTestCommandConfig = 0 THEN
		AssertTrue(Condition := FALSE, Message := 'TEST FAILED: iTestCommandConfig interface is null');
		SequenceCycles := 0;
		RETURN;
	END_IF

	IF iTestComponent = 0 THEN
		AssertTrue(Condition := FALSE, Message := 'TEST FAILED: iTestComponent interface is null');
		SequenceCycles := 0;
		RETURN;
	END_IF

	// Configure command with sequencer callback completion condition
	CompletionCondition	:= (SequenceCycles >= 5);
	iTestCommandConfig.P_CommandConfiguration.CompletionCondition REF= CompletionCondition;
	iTestCommandConfig.P_CommandConfiguration.CommandDescription := 'Sequencer callback test - operation sequencer';
	iTestCommandConfig.P_CommandConfiguration.TimeoutTime := T#5S;
	IF __ISVALIDREF(iTestCommandConfig.P_CommandConfiguration.BaseConfiguration) THEN
		iTestCommandConfig.P_CommandConfiguration.BaseConfiguration.LogTraceConfiguration.When := E_LogTraceWhen.xRunOnInitOnly;
	END_IF

	// Setup component to be enabled and not busy
	IF iTestComponent <> 0 THEN
		iTestComponent.P_ComponentStatus.BaseStatus.Enabled := TRUE;
		iTestComponent.P_ComponentStatus.BaseStatus.Busy := FALSE;
		iTestComponent.P_ComponentStatus.BaseStatus.Error := FALSE;
	END_IF

	// Configure permissive to be OK
	IF iTestPermIntlkConfig <> 0 THEN
		iTestPermIntlkConfig.P_PermIntlkConfiguration.PermIntlkObj[1].Description := 'Sequencer Callback Permissive';
		iTestPermIntlkConfig.P_PermIntlkConfiguration.PermIntlkObj[1].Condition := TRUE;
		iTestPermIntlkConfig.P_PermIntlkConfiguration.PermIntlkObj[1].Index := 1;
		TestPermIntlk[TestIdx].CyclicLogic(); // Update permissive evaluation
	END_IF

	// Setup command with configurations
	iTestCommand.InjectConfigurations(
		iComponent := iTestComponent,
		iCommandConfiguration := iTestCommandConfig,
		iPermIntlkConfiguration := iTestPermIntlkConfig
	);

	// Resolve configurations after injection
	iTestCommand.CyclicLogic();

	// Execute command
	iTestCommand.Execute();

	// Verify Execute() accepted the command
	AssertEquals_UDINT(
		Expected := E_CommandResult.Accepted,
		Actual := iTestCommand.P_CommandStatus.Result,
		Message := 'Execute() should set Result to Accepted'
	);

	SimulatedSequenceStep := 1; // Sequencer at step 1, waiting for command completion
ELSE
	// Refresh interface references for subsequent cycles
	iTestCommand := TestCommand[TestIdx];
	iTestCommandConfig := TestCommandConfig[TestIdx];

	// CRITICAL: Validate interfaces on every cycle to prevent page faults
	IF iTestCommand = 0 OR iTestCommandConfig = 0 THEN
		// Interface became invalid - reset test
		SequenceCycles := 0;
		SimulatedSequenceStep := 0;
		RETURN;
	END_IF
END_IF

SequenceCycles := SequenceCycles + 1;

// Update completion condition dynamically
CompletionCondition	:= (SequenceCycles >= 5);
iTestCommandConfig.P_CommandConfiguration.CompletionCondition ref= CompletionCondition;

// Run cyclic logic
iTestCommand.CyclicLogic();

// When command completes, simulate sequencer advancing to next step
IF iTestCommand.P_CommandStatus.BaseStatus.Done AND SimulatedSequenceStep = 1 THEN
	SimulatedSequenceStep := 2; // Advance to next step (simulating sequencer callback)
END_IF

IF SequenceCycles >= 6 THEN
	AssertEquals_INT(
		Expected := 2,
		Actual := SimulatedSequenceStep,
		Message := 'Sequencer should advance to next step when command completes (callback mechanism)'
	);

	AssertTrue(
		Condition := iTestCommand.P_CommandStatus.BaseStatus.Done,
		Message := 'Command should have Done=TRUE to trigger sequencer callback'
	);

	TEST_FINISHED();
	SequenceCycles := 0;
	SimulatedSequenceStep := 0;
END_IF
END_METHOD

METHOD PRIVATE TEST_CompletionConditionEvaluation
VAR_INST
	EvaluationCount : INT := 0;
	CompletionCondition	: bool;
END_VAR
VAR
	TestName : Tc2_System.T_MaxString := 'TEST_CompletionConditionEvaluation';
	TestIdx : DINT := INDEX_COMPLETIONCONDITIONEVALUATION;
END_VAR
TEST(__POUNAME());

// Initialize test objects on first evaluation only
IF EvaluationCount = 0 THEN
	TestCommand[TestIdx].Initialize();
	TestComponent[TestIdx].Initialize();
	TestCommandConfig[TestIdx].Initialize();
	TestPermIntlk[TestIdx].Initialize();

	// Safe interface assignments
	iTestCommand := TestCommand[TestIdx];
	iTestCommandConfig := TestCommandConfig[TestIdx];
	iTestComponent := TestComponent[TestIdx];
	iTestPermIntlkConfig := TestPermIntlk[TestIdx];

	// Interface validation with protection
	IF iTestCommand = 0 THEN
		AssertTrue(Condition := FALSE, Message := 'TEST FAILED: iTestCommand interface is null');
		EvaluationCount := 0;
		RETURN;
	END_IF

	IF iTestCommandConfig = 0 THEN
		AssertTrue(Condition := FALSE, Message := 'TEST FAILED: iTestCommandConfig interface is null');
		EvaluationCount := 0;
		RETURN;
	END_IF

	IF iTestComponent = 0 THEN
		AssertTrue(Condition := FALSE, Message := 'TEST FAILED: iTestComponent interface is null');
		EvaluationCount := 0;
		RETURN;
	END_IF

	// Configure command with dynamic completion condition (starts FALSE)
	CompletionCondition	:= (EvaluationCount >= 10);
	iTestCommandConfig.P_CommandConfiguration.CompletionCondition REF= CompletionCondition;
	iTestCommandConfig.P_CommandConfiguration.CommandDescription := 'Continuous evaluation test - dynamic condition';
	iTestCommandConfig.P_CommandConfiguration.TimeoutTime := T#30S;
	IF __ISVALIDREF(iTestCommandConfig.P_CommandConfiguration.BaseConfiguration) THEN
		iTestCommandConfig.P_CommandConfiguration.BaseConfiguration.LogTraceConfiguration.When := E_LogTraceWhen.xRunOnInitOnly;
	END_IF

	// Setup component to be enabled and not busy
	IF iTestComponent <> 0 THEN
		iTestComponent.P_ComponentStatus.BaseStatus.Enabled := TRUE;
		iTestComponent.P_ComponentStatus.BaseStatus.Busy := FALSE;
		iTestComponent.P_ComponentStatus.BaseStatus.Error := FALSE;
	END_IF

	// Configure permissive to be OK
	IF iTestPermIntlkConfig <> 0 THEN
		iTestPermIntlkConfig.P_PermIntlkConfiguration.PermIntlkObj[1].Description := 'Evaluation Permissive';
		iTestPermIntlkConfig.P_PermIntlkConfiguration.PermIntlkObj[1].Condition := TRUE;
		iTestPermIntlkConfig.P_PermIntlkConfiguration.PermIntlkObj[1].Index := 1;
		TestPermIntlk[TestIdx].CyclicLogic(); // Update permissive evaluation
	END_IF

	// Setup command with configurations
	iTestCommand.InjectConfigurations(
		iComponent := iTestComponent,
		iCommandConfiguration := iTestCommandConfig,
		iPermIntlkConfiguration := iTestPermIntlkConfig
	);

	// Resolve configurations after injection
	iTestCommand.CyclicLogic();

	// Execute command
	iTestCommand.Execute();

	// Verify Execute() accepted the command
	AssertEquals_UDINT(
		Expected := E_CommandResult.Accepted,
		Actual := iTestCommand.P_CommandStatus.Result,
		Message := 'Execute() should set Result to Accepted'
	);
ELSE
	// Refresh interface references for subsequent evaluations
	iTestCommand := TestCommand[TestIdx];
	iTestCommandConfig := TestCommandConfig[TestIdx];
END_IF

EvaluationCount := EvaluationCount + 1;

// Update completion condition dynamically based on evaluation count BEFORE calling CyclicLogic
iTestCommandConfig.P_CommandConfiguration.CompletionCondition := (EvaluationCount >= 10);

// Run cyclic logic each evaluation
iTestCommand.CyclicLogic();

// Verify command stays in Monitor state while waiting for condition
IF EvaluationCount > 3 AND EvaluationCount < 10 THEN
	AssertEquals_UDINT(
		Expected := E_CommandState.Monitor,
		Actual := iTestCommand.P_CommandStatus.StepState,
		Message := 'Command should stay in Monitor state while continuous evaluation condition is FALSE'
	);

	AssertFalse(
		Condition := iTestCommand.P_CommandStatus.BaseStatus.Done,
		Message := 'Command should not be Done while evaluation condition is not met'
	);
END_IF

// After 11 evaluations, verify command completed (before auto-reset at cycle 3)
IF EvaluationCount >= 11 THEN
	AssertEquals_UDINT(
		Expected := E_CommandState.Complete,
		Actual := iTestCommand.P_CommandStatus.StepState,
		Message := 'Command should be in Complete state after evaluation condition is met'
	);

	AssertTrue(
		Condition := iTestCommand.P_CommandStatus.BaseStatus.Done,
		Message := 'Command should have Done=TRUE when evaluation condition is met (EvaluationCount >= 10)'
	);

	AssertEquals_UDINT(
		Expected := E_CommandResult.Ok,
		Actual := iTestCommand.P_CommandStatus.Result,
		Message := 'Command should have Result=Ok after successful completion'
	);

	TEST_FINISHED();
	EvaluationCount := 0;
END_IF
END_METHOD

METHOD PRIVATE TEST_CompletionWithInterlockDrop
VAR_INST
	TestCycles : INT := 0;
	CompletionCondition	: bool;
END_VAR
VAR
	TestName : Tc2_System.T_MaxString := 'TEST_CompletionWithInterlockDrop';
	TestIdx : DINT := INDEX_COMPLETIONWITHINTERLOCKDROP;
END_VAR
TEST(__POUNAME());

// Initialize test objects on first cycle only
IF TestCycles = 0 THEN
	TestCommand[TestIdx].Initialize();
	TestComponent[TestIdx].Initialize();
	TestCommandConfig[TestIdx].Initialize();
	TestPermIntlk[TestIdx].Initialize();

	// Safe interface assignments
	iTestCommand := TestCommand[TestIdx];
	iTestCommandConfig := TestCommandConfig[TestIdx];
	iTestComponent := TestComponent[TestIdx];
	iTestPermIntlkConfig := TestPermIntlk[TestIdx];

	// Interface validation with protection
	IF iTestCommand = 0 THEN
		AssertTrue(Condition := FALSE, Message := 'TEST FAILED: iTestCommand interface is null');
		TestCycles := 0;
		RETURN;
	END_IF

	IF iTestCommandConfig = 0 THEN
		AssertTrue(Condition := FALSE, Message := 'TEST FAILED: iTestCommandConfig interface is null');
		TestCycles := 0;
		RETURN;
	END_IF

	IF iTestComponent = 0 THEN
		AssertTrue(Condition := FALSE, Message := 'TEST FAILED: iTestComponent interface is null');
		TestCycles := 0;
		RETURN;
	END_IF

	IF iTestPermIntlkConfig = 0 THEN
		AssertTrue(Condition := FALSE, Message := 'TEST FAILED: iTestPermIntlkConfig interface is null');
		TestCycles := 0;
		RETURN;
	END_IF

	// Configure command with completion condition (will become TRUE at cycle 10)
	CompletionCondition	:= (TestCycles >= 10);
	iTestCommandConfig.P_CommandConfiguration.CompletionCondition ref= CompletionCondition;
	iTestCommandConfig.P_CommandConfiguration.AbortOnInterlockDrop := TRUE; // Critical: abort when interlock drops
	iTestCommandConfig.P_CommandConfiguration.PermIntlkConfiguredAsInterlock := TRUE; // Configure as interlock
	iTestCommandConfig.P_CommandConfiguration.CommandDescription := 'Interlock drop during completion evaluation';
	iTestCommandConfig.P_CommandConfiguration.TimeoutTime := T#30S;
	IF __ISVALIDREF(iTestCommandConfig.P_CommandConfiguration.BaseConfiguration) THEN
		iTestCommandConfig.P_CommandConfiguration.BaseConfiguration.LogTraceConfiguration.When := E_LogTraceWhen.xRunOnInitOnly;
	END_IF

	// Setup component to be enabled and not busy
	IF iTestComponent <> 0 THEN
		iTestComponent.P_ComponentStatus.BaseStatus.Enabled := TRUE;
		iTestComponent.P_ComponentStatus.BaseStatus.Busy := FALSE;
		iTestComponent.P_ComponentStatus.BaseStatus.Error := FALSE;
	END_IF

	// Configure permissive/interlock that will drop at cycle 5
	IF iTestPermIntlkConfig <> 0 THEN
		iTestPermIntlkConfig.P_PermIntlkConfiguration.PermIntlkObj[1].Description := 'Dynamic Interlock - Drops at cycle 5';
		iTestPermIntlkConfig.P_PermIntlkConfiguration.PermIntlkObj[1].Condition := (TestCycles < 5); // TRUE until cycle 5
		iTestPermIntlkConfig.P_PermIntlkConfiguration.PermIntlkObj[1].Index := 1;
		TestPermIntlk[TestIdx].CyclicLogic(); // Initialize permissive evaluation
	END_IF

	// Setup command with configurations
	iTestCommand.InjectConfigurations(
		iComponent := iTestComponent,
		iCommandConfiguration := iTestCommandConfig,
		iPermIntlkConfiguration := iTestPermIntlkConfig
	);

	// Resolve configurations after injection
	iTestCommand.CyclicLogic();

	// Execute command
	iTestCommand.Execute();

	// Verify Execute() accepted the command
	AssertEquals_UDINT(
		Expected := E_CommandResult.Accepted,
		Actual := iTestCommand.P_CommandStatus.Result,
		Message := 'Execute() should set Result to Accepted'
	);
ELSE
	// Refresh interface references for subsequent cycles
	iTestCommand := TestCommand[TestIdx];
	iTestCommandConfig := TestCommandConfig[TestIdx];
	iTestPermIntlkConfig := TestPermIntlk[TestIdx];

	// Update dynamic completion condition
	iTestCommandConfig.P_CommandConfiguration.CompletionCondition := (TestCycles >= 10);

	// Update dynamic interlock condition (will drop at cycle 5)
	IF iTestPermIntlkConfig <> 0 THEN
		iTestPermIntlkConfig.P_PermIntlkConfiguration.PermIntlkObj[1].Condition := (TestCycles < 5);
		TestPermIntlk[TestIdx].CyclicLogic(); // Update permissive evaluation
	END_IF
END_IF

// Run cyclic logic and increment counter
iTestCommand.CyclicLogic();
TestCycles := TestCycles + 1;

// At cycle 7, verify command aborted due to interlock drop at cycle 5
IF TestCycles = 7 THEN
	AssertEquals_UDINT(
		Expected := E_CommandResult.InterlockLost,
		Actual := iTestCommand.P_CommandStatus.Result,
		Message := 'Command should abort with InterlockLost when interlock drops during completion evaluation'
	);

	AssertTrue(
		Condition := iTestCommand.P_CommandStatus.BaseStatus.Error,
		Message := 'Command should have Error=TRUE after interlock drop'
	);

	AssertEquals_UDINT(
		Expected := E_CommandState.Complete,
		Actual := iTestCommand.P_CommandStatus.StepState,
		Message := 'Command should be in Complete state after abort due to interlock drop'
	);

	TEST_FINISHED();
	TestCycles := 0;
END_IF
END_METHOD

METHOD PRIVATE TEST_DiscreteCompletionCondition
VAR_INST
	SimulatedOutput : BOOL := FALSE;
	TargetState : BOOL := TRUE;
	DiscreteCycles : INT := 0;
	CompletionCondition	: BOOL;
END_VAR
VAR
	TestName : Tc2_System.T_MaxString := 'TEST_DiscreteCompletionCondition';
	TestIdx : DINT := INDEX_DISCRETECOMPLETIONCONDITION;
END_VAR
TEST(__POUNAME());

// Initialize test objects on first cycle only
IF DiscreteCycles = 0 THEN
	TestCommand[TestIdx].Initialize();
	TestComponent[TestIdx].Initialize();
	TestCommandConfig[TestIdx].Initialize();
	TestPermIntlk[TestIdx].Initialize();

	// Safe interface assignments
	iTestCommand := TestCommand[TestIdx];
	iTestCommandConfig := TestCommandConfig[TestIdx];
	iTestComponent := TestComponent[TestIdx];
	iTestPermIntlkConfig := TestPermIntlk[TestIdx];

	// Interface validation with protection
	IF iTestCommand = 0 THEN
		AssertTrue(Condition := FALSE, Message := 'TEST FAILED: iTestCommand interface is null');
		DiscreteCycles := 0;
		RETURN;
	END_IF

	IF iTestCommandConfig = 0 THEN
		AssertTrue(Condition := FALSE, Message := 'TEST FAILED: iTestCommandConfig interface is null');
		DiscreteCycles := 0;
		RETURN;
	END_IF

	IF iTestComponent = 0 THEN
		AssertTrue(Condition := FALSE, Message := 'TEST FAILED: iTestComponent interface is null');
		DiscreteCycles := 0;
		RETURN;
	END_IF

	// Initialize discrete output simulation
	SimulatedOutput := FALSE;
	TargetState := TRUE;

	// Configure command with discrete output completion condition
	CompletionCondition	:= (SimulatedOutput = TargetState);
	iTestCommandConfig.P_CommandConfiguration.CompletionCondition ref= CompletionCondition;
	iTestCommandConfig.P_CommandConfiguration.CommandDescription := 'Set discrete output - digital IO';
	iTestCommandConfig.P_CommandConfiguration.TimeoutTime := T#5S;
	IF __ISVALIDREF(iTestCommandConfig.P_CommandConfiguration.BaseConfiguration) THEN
		iTestCommandConfig.P_CommandConfiguration.BaseConfiguration.LogTraceConfiguration.When := E_LogTraceWhen.xRunOnInitOnly;
	END_IF

	// Setup component to be enabled and not busy
	IF iTestComponent <> 0 THEN
		iTestComponent.P_ComponentStatus.BaseStatus.Enabled := TRUE;
		iTestComponent.P_ComponentStatus.BaseStatus.Busy := FALSE;
		iTestComponent.P_ComponentStatus.BaseStatus.Error := FALSE;
	END_IF

	// Configure permissive to be OK
	IF iTestPermIntlkConfig <> 0 THEN
		iTestPermIntlkConfig.P_PermIntlkConfiguration.PermIntlkObj[1].Description := 'Discrete Completion Permissive';
		iTestPermIntlkConfig.P_PermIntlkConfiguration.PermIntlkObj[1].Condition := TRUE;
		iTestPermIntlkConfig.P_PermIntlkConfiguration.PermIntlkObj[1].Index := 1;
		TestPermIntlk[TestIdx].CyclicLogic(); // Update permissive evaluation
	END_IF

	// Setup command with configurations
	iTestCommand.InjectConfigurations(
		iComponent := iTestComponent,
		iCommandConfiguration := iTestCommandConfig,
		iPermIntlkConfiguration := iTestPermIntlkConfig
	);

	// Resolve configurations after injection
	iTestCommand.CyclicLogic();

	// Execute command
	iTestCommand.Execute();

	// Verify Execute() accepted the command
	AssertEquals_UDINT(
		Expected := E_CommandResult.Accepted,
		Actual := iTestCommand.P_CommandStatus.Result,
		Message := 'Execute() should set Result to Accepted'
	);
ELSE
	// Refresh interface references for subsequent cycles
	iTestCommand := TestCommand[TestIdx];
	iTestCommandConfig := TestCommandConfig[TestIdx];

	// CRITICAL: Validate interfaces on every cycle to prevent page faults
	IF iTestCommand = 0 OR iTestCommandConfig = 0 THEN
		// Interface became invalid - reset test
		DiscreteCycles := 0;
		SimulatedOutput := FALSE;
		RETURN;
	END_IF
END_IF

DiscreteCycles := DiscreteCycles + 1;

// Simulate discrete output changing state after 3 cycles
IF DiscreteCycles = 3 THEN
	SimulatedOutput := TRUE;
END_IF

// Update completion condition dynamically based on simulated output
iTestCommandConfig.P_CommandConfiguration.CompletionCondition := (SimulatedOutput = TargetState);

// Run cyclic logic
iTestCommand.CyclicLogic();

// Check completion after output reaches target state
IF DiscreteCycles >= 5 THEN
	AssertEquals_UDINT(
		Expected := E_CommandState.Complete,
		Actual := iTestCommand.P_CommandStatus.StepState,
		Message := 'Discrete command should be in Complete state when output matches target state'
	);

	AssertTrue(
		Condition := iTestCommand.P_CommandStatus.BaseStatus.Done,
		Message := 'Discrete command should have Done=TRUE when output matches target state'
	);

	AssertEquals_UDINT(
		Expected := E_CommandResult.Ok,
		Actual := iTestCommand.P_CommandStatus.Result,
		Message := 'Discrete command should have Result=Ok after output state matches target'
	);

	TEST_FINISHED();
	SimulatedOutput := FALSE;
	DiscreteCycles := 0;
END_IF
END_METHOD

METHOD PRIVATE TEST_DynamicCompletionConditionUpdate
VAR_INST
	DynamicCycles : INT := 0;
	TargetValue : INT := 5;
	CompletionCondition	: BOOL;
END_VAR
VAR
	TestName : Tc2_System.T_MaxString := 'TEST_DynamicCompletionConditionUpdate';
	TestIdx : DINT := INDEX_DYNAMICCOMPLETIONCONDITIONUPDATE;
END_VAR
TEST(__POUNAME());

// Initialize test objects on first cycle only
IF DynamicCycles = 0 THEN
	TestCommand[TestIdx].Initialize();
	TestComponent[TestIdx].Initialize();
	TestCommandConfig[TestIdx].Initialize();
	TestPermIntlk[TestIdx].Initialize();

	// Safe interface assignments
	iTestCommand := TestCommand[TestIdx];
	iTestCommandConfig := TestCommandConfig[TestIdx];
	iTestComponent := TestComponent[TestIdx];
	iTestPermIntlkConfig := TestPermIntlk[TestIdx];

	// Interface validation with protection
	IF iTestCommand = 0 THEN
		AssertTrue(Condition := FALSE, Message := 'TEST FAILED: iTestCommand interface is null');
		DynamicCycles := 0;
		RETURN;
	END_IF

	IF iTestCommandConfig = 0 THEN
		AssertTrue(Condition := FALSE, Message := 'TEST FAILED: iTestCommandConfig interface is null');
		DynamicCycles := 0;
		RETURN;
	END_IF

	IF iTestComponent = 0 THEN
		AssertTrue(Condition := FALSE, Message := 'TEST FAILED: iTestComponent interface is null');
		DynamicCycles := 0;
		RETURN;
	END_IF

	// Configure command with initial dynamic completion condition
	TargetValue := 5;
	CompletionCondition	:= (DynamicCycles >= TargetValue);
	iTestCommandConfig.P_CommandConfiguration.CompletionCondition REF= CompletionCondition; 
	iTestCommandConfig.P_CommandConfiguration.CommandDescription := 'Dynamic condition update test - Recipe Manager';
	iTestCommandConfig.P_CommandConfiguration.TimeoutTime := T#30S;
	IF __ISVALIDREF(iTestCommandConfig.P_CommandConfiguration.BaseConfiguration) THEN
		iTestCommandConfig.P_CommandConfiguration.BaseConfiguration.LogTraceConfiguration.When := E_LogTraceWhen.xRunOnInitOnly;
	END_IF

	// Setup component to be enabled and not busy
	IF iTestComponent <> 0 THEN
		iTestComponent.P_ComponentStatus.BaseStatus.Enabled := TRUE;
		iTestComponent.P_ComponentStatus.BaseStatus.Busy := FALSE;
		iTestComponent.P_ComponentStatus.BaseStatus.Error := FALSE;
	END_IF

	// Configure permissive to be OK
	IF iTestPermIntlkConfig <> 0 THEN
		iTestPermIntlkConfig.P_PermIntlkConfiguration.PermIntlkObj[1].Description := 'Dynamic Update Permissive';
		iTestPermIntlkConfig.P_PermIntlkConfiguration.PermIntlkObj[1].Condition := TRUE;
		iTestPermIntlkConfig.P_PermIntlkConfiguration.PermIntlkObj[1].Index := 1;
		TestPermIntlk[TestIdx].CyclicLogic(); // Update permissive evaluation
	END_IF

	// Setup command with configurations
	iTestCommand.InjectConfigurations(
		iComponent := iTestComponent,
		iCommandConfiguration := iTestCommandConfig,
		iPermIntlkConfiguration := iTestPermIntlkConfig
	);

	// Resolve configurations after injection
	iTestCommand.CyclicLogic();

	// Execute command
	iTestCommand.Execute();

	// Verify Execute() accepted the command
	AssertEquals_UDINT(
		Expected := E_CommandResult.Accepted,
		Actual := iTestCommand.P_CommandStatus.Result,
		Message := 'Execute() should set Result to Accepted'
	);
ELSE
	// Refresh interface references for subsequent cycles
	iTestCommand := TestCommand[TestIdx];
	iTestCommandConfig := TestCommandConfig[TestIdx];
END_IF

DynamicCycles := DynamicCycles + 1;

// Change target mid-execution (simulating Recipe Manager dynamically updating condition)
IF DynamicCycles = 3 THEN
	TargetValue := 8; // Extend the target during execution
END_IF

// Update completion condition dynamically
CompletionCondition	:= (DynamicCycles >= TargetValue);
iTestCommandConfig.P_CommandConfiguration.CompletionCondition REF= CompletionCondition; 

// Run cyclic logic
iTestCommand.CyclicLogic();

// Check that command completes with dynamically updated target
IF DynamicCycles >= 10 THEN
	AssertTrue(
		Condition := iTestCommand.P_CommandStatus.BaseStatus.Done,
		Message := 'Command should complete with dynamically updated condition from Recipe Manager'
	);

	AssertTrue(
		Condition := DynamicCycles >= 8,
		Message := 'Command should have waited for dynamically updated target value (8 instead of 5)'
	);

	AssertEquals_UDINT(
		Expected := E_CommandResult.Ok,
		Actual := iTestCommand.P_CommandStatus.Result,
		Message := 'Command should have Result=Ok after dynamic completion'
	);

	TEST_FINISHED();
	DynamicCycles := 0;
	TargetValue := 5;
END_IF
END_METHOD

METHOD PRIVATE TEST_FastCompletionInOneScan
VAR
	TestName : Tc2_System.T_MaxString := 'TEST_FastCompletionInOneScan';
	TestIdx : DINT := INDEX_FASTCOMPLETIONINONESCAN;
	CompletionCondition	: BOOL;
END_VAR
TEST(__POUNAME());

// Initialize test objects first
TestCommand[TestIdx].Initialize();
TestComponent[TestIdx].Initialize();
TestCommandConfig[TestIdx].Initialize();
TestPermIntlk[TestIdx].Initialize();

// Safe interface assignments
iTestCommand := TestCommand[TestIdx];
iTestCommandConfig := TestCommandConfig[TestIdx];
iTestComponent := TestComponent[TestIdx];
iTestPermIntlkConfig := TestPermIntlk[TestIdx];

// Interface validation with protection
IF iTestCommand = 0 THEN
	AssertTrue(Condition := FALSE, Message := 'TEST FAILED: iTestCommand interface is null');
	RETURN;
END_IF

IF iTestCommandConfig = 0 THEN
	AssertTrue(Condition := FALSE, Message := 'TEST FAILED: iTestCommandConfig interface is null');
	RETURN;
END_IF

IF iTestComponent = 0 THEN
	AssertTrue(Condition := FALSE, Message := 'TEST FAILED: iTestComponent interface is null');
	RETURN;
END_IF

// Configure command with completion condition immediately TRUE
CompletionCondition	:= TRUE;
iTestCommandConfig.P_CommandConfiguration.CompletionCondition REF= CompletionCondition;
iTestCommandConfig.P_CommandConfiguration.CommandDescription := 'Fast completion test';
iTestCommandConfig.P_CommandConfiguration.TimeoutTime := T#30S;
IF __ISVALIDREF(iTestCommandConfig.P_CommandConfiguration.BaseConfiguration) THEN
	iTestCommandConfig.P_CommandConfiguration.BaseConfiguration.LogTraceConfiguration.When := E_LogTraceWhen.xRunOnInitOnly;
END_IF

// Setup component to be enabled and not busy
IF iTestComponent <> 0 THEN
	iTestComponent.P_ComponentStatus.BaseStatus.Enabled := TRUE;
	iTestComponent.P_ComponentStatus.BaseStatus.Busy := FALSE;
	iTestComponent.P_ComponentStatus.BaseStatus.Error := FALSE;
END_IF

// Configure permissive to be OK
IF iTestPermIntlkConfig <> 0 THEN
	iTestPermIntlkConfig.P_PermIntlkConfiguration.PermIntlkObj[1].Description := 'Fast Completion Permissive';
	iTestPermIntlkConfig.P_PermIntlkConfiguration.PermIntlkObj[1].Condition := TRUE;
	iTestPermIntlkConfig.P_PermIntlkConfiguration.PermIntlkObj[1].Index := 1;
	TestPermIntlk[TestIdx].CyclicLogic(); // Update permissive evaluation
END_IF

// Setup command with configurations
iTestCommand.InjectConfigurations(
	iComponent := iTestComponent,
	iCommandConfiguration := iTestCommandConfig,
	iPermIntlkConfiguration := iTestPermIntlkConfig
);

// Resolve configurations after injection
iTestCommand.CyclicLogic();

// Execute command
iTestCommand.Execute();

// Verify Execute() accepted the command
AssertEquals_UDINT(
	Expected := E_CommandResult.Accepted,
	Actual := iTestCommand.P_CommandStatus.Result,
	Message := 'Execute() should set Result to Accepted'
);

// State machine progression with completion condition TRUE
iTestCommand.CyclicLogic(); // Idle → Execute
AssertEquals_UDINT(
	Expected := E_CommandState.Execute,
	Actual := iTestCommand.P_CommandStatus.StepState,
	Message := 'First CyclicLogic: Idle → Execute'
);

iTestCommand.CyclicLogic(); // Execute → Monitor
AssertEquals_UDINT(
	Expected := E_CommandState.Monitor,
	Actual := iTestCommand.P_CommandStatus.StepState,
	Message := 'Second CyclicLogic: Execute → Monitor'
);

iTestCommand.Complete(); // Signal completion (CompletionCondition is TRUE)
iTestCommand.CyclicLogic(); // Monitor → Complete
AssertEquals_UDINT(
	Expected := E_CommandState.Complete,
	Actual := iTestCommand.P_CommandStatus.StepState,
	Message := 'Third CyclicLogic: Monitor → Complete (fast completion due to CompletionCondition=TRUE)'
);

// Verify completion status
AssertTrue(
	Condition := iTestCommand.P_CommandStatus.BaseStatus.Done,
	Message := 'Command should have Done=TRUE when completion condition is immediately true'
);

AssertEquals_UDINT(
	Expected := E_CommandResult.Ok,
	Actual := iTestCommand.P_CommandStatus.Result,
	Message := 'Command should have Result=Ok in Complete state'
);

AssertFalse(
	Condition := iTestCommand.P_CommandStatus.BaseStatus.Busy,
	Message := 'Command should clear Busy=FALSE in Complete state'
);

TEST_FINISHED();
END_METHOD

METHOD PRIVATE TEST_MotionCompletionCondition
VAR_INST
	SimulatedPosition : LREAL := 0.0;
	MotionCycles : INT := 0;
	CompletionCondition	: BOOL;
END_VAR
VAR
	TestName : Tc2_System.T_MaxString := 'TEST_MotionCompletionCondition';
	TestIdx : DINT := INDEX_MOTIONCOMPLETIONCONDITION;
	TestTargetPosition : LREAL := 100.0;
	TestPositionTolerance : LREAL := 0.1;
END_VAR
TEST(__POUNAME());

// Initialize test objects on first cycle only
IF MotionCycles = 0 THEN
	TestCommand[TestIdx].Initialize();
	TestComponent[TestIdx].Initialize();
	TestCommandConfig[TestIdx].Initialize();
	TestPermIntlk[TestIdx].Initialize();

	// Safe interface assignments
	iTestCommand := TestCommand[TestIdx];
	iTestCommandConfig := TestCommandConfig[TestIdx];
	iTestComponent := TestComponent[TestIdx];
	iTestPermIntlkConfig := TestPermIntlk[TestIdx];

	// Interface validation with protection
	IF iTestCommand = 0 THEN
		AssertTrue(Condition := FALSE, Message := 'TEST FAILED: iTestCommand interface is null');
		MotionCycles := 0;
		RETURN;
	END_IF

	IF iTestCommandConfig = 0 THEN
		AssertTrue(Condition := FALSE, Message := 'TEST FAILED: iTestCommandConfig interface is null');
		MotionCycles := 0;
		RETURN;
	END_IF

	IF iTestComponent = 0 THEN
		AssertTrue(Condition := FALSE, Message := 'TEST FAILED: iTestComponent interface is null');
		MotionCycles := 0;
		RETURN;
	END_IF

	// Initialize motion simulation
	SimulatedPosition := 0.0;

	// Configure command with motion-based completion condition
	CompletionCondition	:= ABS(SimulatedPosition - TestTargetPosition) <= TestPositionTolerance;
	iTestCommandConfig.P_CommandConfiguration.CompletionCondition REF= CompletionCondition;
	iTestCommandConfig.P_CommandConfiguration.CommandDescription := 'Motion to target position - axis positioning';
	iTestCommandConfig.P_CommandConfiguration.TimeoutTime := T#5S;
	IF __ISVALIDREF(iTestCommandConfig.P_CommandConfiguration.BaseConfiguration) THEN
		iTestCommandConfig.P_CommandConfiguration.BaseConfiguration.LogTraceConfiguration.When := E_LogTraceWhen.xRunOnInitOnly;
	END_IF

	// Setup component to be enabled and not busy
	IF iTestComponent <> 0 THEN
		iTestComponent.P_ComponentStatus.BaseStatus.Enabled := TRUE;
		iTestComponent.P_ComponentStatus.BaseStatus.Busy := FALSE;
		iTestComponent.P_ComponentStatus.BaseStatus.Error := FALSE;
	END_IF

	// Configure permissive to be OK
	IF iTestPermIntlkConfig <> 0 THEN
		iTestPermIntlkConfig.P_PermIntlkConfiguration.PermIntlkObj[1].Description := 'Motion Completion Permissive';
		iTestPermIntlkConfig.P_PermIntlkConfiguration.PermIntlkObj[1].Condition := TRUE;
		iTestPermIntlkConfig.P_PermIntlkConfiguration.PermIntlkObj[1].Index := 1;
		TestPermIntlk[TestIdx].CyclicLogic(); // Update permissive evaluation
	END_IF

	// Setup command with configurations
	iTestCommand.InjectConfigurations(
		iComponent := iTestComponent,
		iCommandConfiguration := iTestCommandConfig,
		iPermIntlkConfiguration := iTestPermIntlkConfig
	);

	// Resolve configurations after injection
	iTestCommand.CyclicLogic();

	// Execute command
	iTestCommand.Execute();

	// Verify Execute() accepted the command
	AssertEquals_UDINT(
		Expected := E_CommandResult.Accepted,
		Actual := iTestCommand.P_CommandStatus.Result,
		Message := 'Execute() should set Result to Accepted'
	);
ELSE
	// Refresh interface references for subsequent cycles
	iTestCommand := TestCommand[TestIdx];
	iTestCommandConfig := TestCommandConfig[TestIdx];

	// CRITICAL: Validate interfaces on every cycle to prevent page faults
	IF iTestCommand = 0 OR iTestCommandConfig = 0 THEN
		// Interface became invalid - reset test
		MotionCycles := 0;
		SimulatedPosition := 0.0;
		RETURN;
	END_IF
END_IF

// Simulate motion - move 10 units per cycle toward target
SimulatedPosition := MIN(SimulatedPosition + 10.0, TestTargetPosition);
MotionCycles := MotionCycles + 1;

// Update completion condition dynamically based on simulated position
iTestCommandConfig.P_CommandConfiguration.CompletionCondition := ABS(SimulatedPosition - TestTargetPosition) <= TestPositionTolerance;

// Signal completion when position reaches target
IF ABS(SimulatedPosition - TestTargetPosition) <= TestPositionTolerance THEN
	iTestCommand.Complete();
END_IF

// Run cyclic logic
iTestCommand.CyclicLogic();

// Check completion when position is reached
IF SimulatedPosition >= TestTargetPosition - TestPositionTolerance THEN
	IF MotionCycles > 12 THEN // Allow time for state transitions
		AssertEquals_UDINT(
			Expected := E_CommandState.Complete,
			Actual := iTestCommand.P_CommandStatus.StepState,
			Message := 'Motion command should be in Complete state when position is within tolerance'
		);

		AssertTrue(
			Condition := iTestCommand.P_CommandStatus.BaseStatus.Done,
			Message := 'Motion command should have Done=TRUE when position is within tolerance'
		);

		AssertEquals_UDINT(
			Expected := E_CommandResult.Ok,
			Actual := iTestCommand.P_CommandStatus.Result,
			Message := 'Motion command should have Result=Ok after reaching target position'
		);

		TEST_FINISHED();
		SimulatedPosition := 0.0;
		MotionCycles := 0;
	END_IF
END_IF
END_METHOD

METHOD PRIVATE TEST_OperationToCommandTranslation
VAR
	TestName : Tc2_System.T_MaxString := 'TEST_OperationToCommandTranslation';
	TestIdx : DINT := INDEX_OPERATIONTOCOMMANDTRANSLATION;
	TestOp : ST_Operation;
	CompletionCondition	: BOOL;
END_VAR
TEST(__POUNAME());

// This test verifies mapping from ST_Operation to ST_CommandConfiguration
// Tests translation layer between operation sequencer and command execution

// Initialize test objects first
TestCommand[TestIdx].Initialize();
TestComponent[TestIdx].Initialize();
TestCommandConfig[TestIdx].Initialize();
TestPermIntlk[TestIdx].Initialize();

// Safe interface assignments
iTestCommand := TestCommand[TestIdx];
iTestCommandConfig := TestCommandConfig[TestIdx];
iTestComponent := TestComponent[TestIdx];
iTestPermIntlkConfig := TestPermIntlk[TestIdx];

// Interface validation with protection
IF iTestCommand = 0 THEN
	AssertTrue(Condition := FALSE, Message := 'TEST FAILED: iTestCommand interface is null');
	RETURN;
END_IF

IF iTestCommandConfig = 0 THEN
	AssertTrue(Condition := FALSE, Message := 'TEST FAILED: iTestCommandConfig interface is null');
	RETURN;
END_IF

IF iTestComponent = 0 THEN
	AssertTrue(Condition := FALSE, Message := 'TEST FAILED: iTestComponent interface is null');
	RETURN;
END_IF

// Setup: Create an operation structure (simulating operation sequencer input)
TestOp.OperationID := E_Operation.Wait;
TestOp.Timeout := T#3S;
TestOp.HMILabel := 'Wait operation';

// Translate ST_Operation to ST_CommandConfiguration (this is the mapping logic being tested)
iTestCommandConfig.P_CommandConfiguration.CommandIndex := TestOp.OperationID;
iTestCommandConfig.P_CommandConfiguration.TimeoutTime := TestOp.Timeout;
iTestCommandConfig.P_CommandConfiguration.CommandDescription := TestOp.HMILabel;
CompletionCondition	:= FALSE;
iTestCommandConfig.P_CommandConfiguration.CompletionCondition REF= CompletionCondition; // Will be set based on operation type
IF __ISVALIDREF(iTestCommandConfig.P_CommandConfiguration.BaseConfiguration) THEN
	iTestCommandConfig.P_CommandConfiguration.BaseConfiguration.LogTraceConfiguration.When := E_LogTraceWhen.xRunOnInitOnly;
END_IF

// Setup component to be enabled and not busy
IF iTestComponent <> 0 THEN
	iTestComponent.P_ComponentStatus.BaseStatus.Enabled := TRUE;
	iTestComponent.P_ComponentStatus.BaseStatus.Busy := FALSE;
	iTestComponent.P_ComponentStatus.BaseStatus.Error := FALSE;
END_IF

// Configure permissive to be OK
IF iTestPermIntlkConfig <> 0 THEN
	iTestPermIntlkConfig.P_PermIntlkConfiguration.PermIntlkObj[1].Description := 'Operation Translation Permissive';
	iTestPermIntlkConfig.P_PermIntlkConfiguration.PermIntlkObj[1].Condition := TRUE;
	iTestPermIntlkConfig.P_PermIntlkConfiguration.PermIntlkObj[1].Index := 1;
END_IF

// Inject configurations
iTestCommand.InjectConfigurations(
	iComponent := iTestComponent,
	iCommandConfiguration := iTestCommandConfig,
	iPermIntlkConfiguration := iTestPermIntlkConfig
);

// Resolve configurations after injection
iTestCommand.CyclicLogic();

// Verify translation from ST_Operation to ST_CommandConfiguration
AssertEquals_DINT(
	Expected := E_Operation.Wait,
	Actual := iTestCommandConfig.P_CommandConfiguration.CommandIndex,
	Message := 'Command CommandIndex should match ST_Operation.OperationID after translation'
);

AssertEquals_STRING(
	Expected := 'Wait operation',
	Actual := iTestCommandConfig.P_CommandConfiguration.CommandDescription,
	Message := 'Command CommandDescription should match ST_Operation.HMILabel after translation'
);

AssertEquals_TIME(
	Expected := T#3S,
	Actual := iTestCommandConfig.P_CommandConfiguration.TimeoutTime,
	Message := 'Command TimeoutTime should match ST_Operation.Timeout after translation'
);

TEST_FINISHED();
END_METHOD

METHOD PRIVATE TEST_RecipeManagerProvidesCommandConfig
VAR
	TestName : Tc2_System.T_MaxString := 'TEST_RecipeManagerProvidesCommandConfig';
	TestIdx : DINT := INDEX_RECIPEMANAGERPROVIDESCOMMANDCONFIG;
	CompletionCondition	: BOOL;
END_VAR
TEST(__POUNAME());

// This test verifies that command configurations can be dynamically provided by Recipe Manager
// Simulates external system (Recipe Manager) injecting command configuration at runtime

// Initialize test objects first
TestCommand[TestIdx].Initialize();
TestComponent[TestIdx].Initialize();
TestCommandConfig[TestIdx].Initialize();
TestPermIntlk[TestIdx].Initialize();

// Safe interface assignments
iTestCommand := TestCommand[TestIdx];
iTestCommandConfig := TestCommandConfig[TestIdx];
iTestComponent := TestComponent[TestIdx];
iTestPermIntlkConfig := TestPermIntlk[TestIdx];

// Interface validation with protection
IF iTestCommand = 0 THEN
	AssertTrue(Condition := FALSE, Message := 'TEST FAILED: iTestCommand interface is null');
	RETURN;
END_IF

IF iTestCommandConfig = 0 THEN
	AssertTrue(Condition := FALSE, Message := 'TEST FAILED: iTestCommandConfig interface is null');
	RETURN;
END_IF

IF iTestComponent = 0 THEN
	AssertTrue(Condition := FALSE, Message := 'TEST FAILED: iTestComponent interface is null');
	RETURN;
END_IF

// Setup: Simulate Recipe Manager dynamically setting command configuration
iTestCommandConfig.P_CommandConfiguration.CommandDescription := 'Recipe-provided command';
iTestCommandConfig.P_CommandConfiguration.TimeoutTime := T#5S;
iTestCommandConfig.P_CommandConfiguration.Priority := E_CommandPriority.Priority_High;
CompletionCondition	:= TRUE;
iTestCommandConfig.P_CommandConfiguration.CompletionCondition REF= CompletionCondition; // Fast completion for test
IF __ISVALIDREF(iTestCommandConfig.P_CommandConfiguration.BaseConfiguration) THEN
	iTestCommandConfig.P_CommandConfiguration.BaseConfiguration.LogTraceConfiguration.When := E_LogTraceWhen.xRunOnInitOnly;
END_IF

// Setup component to be enabled and not busy
IF iTestComponent <> 0 THEN
	iTestComponent.P_ComponentStatus.BaseStatus.Enabled := TRUE;
	iTestComponent.P_ComponentStatus.BaseStatus.Busy := FALSE;
	iTestComponent.P_ComponentStatus.BaseStatus.Error := FALSE;
END_IF

// Configure permissive to be OK
IF iTestPermIntlkConfig <> 0 THEN
	iTestPermIntlkConfig.P_PermIntlkConfiguration.PermIntlkObj[1].Description := 'Recipe Manager Permissive';
	iTestPermIntlkConfig.P_PermIntlkConfiguration.PermIntlkObj[1].Condition := TRUE;
	iTestPermIntlkConfig.P_PermIntlkConfiguration.PermIntlkObj[1].Index := 1;
END_IF

// Inject configurations (simulating Recipe Manager providing configuration)
iTestCommand.InjectConfigurations(
	iComponent := iTestComponent,
	iCommandConfiguration := iTestCommandConfig,
	iPermIntlkConfiguration := iTestPermIntlkConfig
);

// Resolve configurations after injection
iTestCommand.CyclicLogic();

// Verify configuration was properly stored and is accessible
AssertEquals_STRING(
	Expected := 'Recipe-provided command',
	Actual := iTestCommandConfig.P_CommandConfiguration.CommandDescription,
	Message := 'Command should use recipe-provided description from external source'
);

AssertEquals_TIME(
	Expected := T#5S,
	Actual := iTestCommandConfig.P_CommandConfiguration.TimeoutTime,
	Message := 'Command should use recipe-provided timeout from external source'
);

AssertEquals_DINT(
	Expected := TO_DINT(E_CommandPriority.Priority_High),
	Actual := TO_DINT(iTestCommandConfig.P_CommandConfiguration.Priority),
	Message := 'Command should use recipe-provided priority from external source'
);

TEST_FINISHED();
END_METHOD

METHOD PRIVATE TEST_TimeBasedCompletionCondition
VAR_INST
	WaitTimer : TON;
	WaitTime : TIME := T#100MS; // Short time for test
	TestStarted : BOOL := FALSE;
	CompletionCondition	: BOOL;
END_VAR
VAR
	TestName : Tc2_System.T_MaxString := 'TEST_TimeBasedCompletionCondition';
	TestIdx : DINT := INDEX_TIMEBASEDCOMPLETIONCONDITION;
END_VAR
TEST(__POUNAME());

// Initialize test objects on first run only
IF NOT TestStarted THEN
	TestCommand[TestIdx].Initialize();
	TestComponent[TestIdx].Initialize();
	TestCommandConfig[TestIdx].Initialize();
	TestPermIntlk[TestIdx].Initialize();

	// Safe interface assignments
	iTestCommand := TestCommand[TestIdx];
	iTestCommandConfig := TestCommandConfig[TestIdx];
	iTestComponent := TestComponent[TestIdx];
	iTestPermIntlkConfig := TestPermIntlk[TestIdx];

	// Interface validation with protection
	IF iTestCommand = 0 THEN
		AssertTrue(Condition := FALSE, Message := 'TEST FAILED: iTestCommand interface is null');
		TestStarted := FALSE;
		RETURN;
	END_IF

	IF iTestCommandConfig = 0 THEN
		AssertTrue(Condition := FALSE, Message := 'TEST FAILED: iTestCommandConfig interface is null');
		TestStarted := FALSE;
		RETURN;
	END_IF

	IF iTestComponent = 0 THEN
		AssertTrue(Condition := FALSE, Message := 'TEST FAILED: iTestComponent interface is null');
		TestStarted := FALSE;
		RETURN;
	END_IF

	// Configure command with time-based completion condition
	CompletionCondition	:= WaitTimer.Q;
	iTestCommandConfig.P_CommandConfiguration.CompletionCondition REF= CompletionCondition; 
	iTestCommandConfig.P_CommandConfiguration.CommandDescription := 'Wait for timer - time-based operation';
	iTestCommandConfig.P_CommandConfiguration.TimeoutTime := T#5S;
	IF __ISVALIDREF(iTestCommandConfig.P_CommandConfiguration.BaseConfiguration) THEN
		iTestCommandConfig.P_CommandConfiguration.BaseConfiguration.LogTraceConfiguration.When := E_LogTraceWhen.xRunOnInitOnly;
	END_IF

	// Setup component to be enabled and not busy
	IF iTestComponent <> 0 THEN
		iTestComponent.P_ComponentStatus.BaseStatus.Enabled := TRUE;
		iTestComponent.P_ComponentStatus.BaseStatus.Busy := FALSE;
		iTestComponent.P_ComponentStatus.BaseStatus.Error := FALSE;
	END_IF

	// Configure permissive to be OK
	IF iTestPermIntlkConfig <> 0 THEN
		iTestPermIntlkConfig.P_PermIntlkConfiguration.PermIntlkObj[1].Description := 'Time-based Completion Permissive';
		iTestPermIntlkConfig.P_PermIntlkConfiguration.PermIntlkObj[1].Condition := TRUE;
		iTestPermIntlkConfig.P_PermIntlkConfiguration.PermIntlkObj[1].Index := 1;
	END_IF

	// Setup command with configurations
	iTestCommand.InjectConfigurations(
		iComponent := iTestComponent,
		iCommandConfiguration := iTestCommandConfig,
		iPermIntlkConfiguration := iTestPermIntlkConfig
	);

	// Resolve configurations after injection
	iTestCommand.CyclicLogic();

	// Execute command
	iTestCommand.Execute();

	// Verify Execute() accepted the command
	AssertEquals_UDINT(
		Expected := E_CommandResult.Accepted,
		Actual := iTestCommand.P_CommandStatus.Result,
		Message := 'Execute() should set Result to Accepted'
	);

	TestStarted := TRUE;
ELSE
	// Refresh interface references for subsequent runs
	iTestCommand := TestCommand[TestIdx];
	iTestCommandConfig := TestCommandConfig[TestIdx];

	// CRITICAL: Validate interfaces on every cycle to prevent page faults
	IF iTestCommand = 0 OR iTestCommandConfig = 0 THEN
		// Interface became invalid - reset test
		TestStarted := FALSE;
		WaitTimer(IN := FALSE);
		RETURN;
	END_IF
END_IF

// Run wait timer for time-based completion
WaitTimer(IN := TRUE, PT := WaitTime);

// Update completion condition dynamically based on timer state
CompletionCondition	:= WaitTimer.Q;
iTestCommandConfig.P_CommandConfiguration.CompletionCondition REF= CompletionCondition;

// Run cyclic logic
iTestCommand.CyclicLogic();

// Check that command completes when timer expires
IF WaitTimer.Q THEN
	AssertEquals_UDINT(
		Expected := E_CommandState.Complete,
		Actual := iTestCommand.P_CommandStatus.StepState,
		Message := 'Time-based command should be in Complete state when timer expires'
	);

	AssertTrue(
		Condition := iTestCommand.P_CommandStatus.BaseStatus.Done,
		Message := 'Time-based command should have Done=TRUE when timer expires'
	);

	AssertEquals_UDINT(
		Expected := E_CommandResult.Ok,
		Actual := iTestCommand.P_CommandStatus.Result,
		Message := 'Time-based command should have Result=Ok after timer completes'
	);

	TEST_FINISHED();
	WaitTimer(IN := FALSE);
	TestStarted := FALSE;
END_IF
END_METHOD

END_FUNCTION_BLOCK

// Tests/FB_CommandTestsIII
FUNCTION_BLOCK FB_CommandTestsIII EXTENDS TcUnit.FB_TestSuite
VAR CONSTANT
	// Test method index constants - one unique index per test method (0-113)

	// GivenCommand* helper test methods (0-25)
	INDEX_GIVENCOMMAND_WHENCANCEL_EXPECTREMOVEDFROMQUEUE							: DINT := 0;
	INDEX_GIVENCOMMAND_WHENCYCLICLOGICCALLED_EXPECTUPDATED							: DINT := 1;
	INDEX_GIVENCOMMAND_WHENEXECUTECALLED_EXPECTEXECUTION							: DINT := 2;
	INDEX_GIVENCOMMAND_WHENPAUSECALLED_EXPECTCOMMANDPAUSES							: DINT := 3;
	INDEX_GIVENCOMMAND_WHENQUEUECALLED_EXPECTADDEDTOQUEUE							: DINT := 4;
	INDEX_GIVENCOMMAND_WHENRESETCALLED_EXPECTSTATECLEARED							: DINT := 5;
	INDEX_GIVENCOMMAND_WHENRESUMECALLED_EXPECTCOMMANDRESUMES						: DINT := 6;
	INDEX_GIVENCOMMAND_WHENVALIDATECALLED_EXPECTPERMISSIVEOK						: DINT := 7;
	INDEX_GIVENCOMMAND_WHENVALIDATECALLED_EXPECTMATCHCONFIG							: DINT := 8;
	INDEX_GIVENCOMMANDALREADYRUNNING_WHENEXECUTE_CONFLICT							: DINT := 9;
	INDEX_GIVENCOMMANDEXECUTED_WHENCYCLICLOGICRUNS_EXPECTSTATEPROGRESSION			: DINT := 10;
	INDEX_GIVENCOMMANDINIDLESTATE_WHENCANCEL_EXPECTNOACTIONTAKEN					: DINT := 11;
	INDEX_GIVENCOMMANDINVALID_WHENVALIDATECALLED_EXPECTFALSE						: DINT := 12;
	INDEX_GIVENCOMMANDPAUSED_WHENABORT_EXPECTCOMMANDABORTEDANDSTATUSUPDATED			: DINT := 13;
	INDEX_GIVENCOMMANDPAUSED_WHENRESUME_EXPECTCOMMANDRESUMESEXECUTION				: DINT := 14;
	INDEX_GIVENCOMMANDQUEUED_WHENABORT_EXPECTCOMMANDABORTEDANDSTATUSUPDATED			: DINT := 15;
	INDEX_GIVENCOMMANDQUEUED_WHENCANCEL_EXPECTCOMMANDREMOVEDFROMQUEUE				: DINT := 16;
	INDEX_GIVENCOMMANDVALIDATED_WHENVALIDATECALLED_EXPECTTRUE						: DINT := 17;
	INDEX_GIVENCOMPONENTRESET_WHENRESETCALLED_EXPECTALLCOMMANDSTATECLEARED			: DINT := 18;
	INDEX_GIVENINJECTEDCONFIGURATIONSVALID_EXPECTINTERFACESSTOREDANDINITIALIZED		: DINT := 19;
	INDEX_GIVENINVALIDCONFIGURATION_WHENINJECTCONFIGURATIONCALLED_EXPECTINITFAILURE	: DINT := 20;
	INDEX_GIVENINVALIDCONFIGURATIONS_WHENINJECTCONFIGURATIONS_EXPECTINITFAILURE		: DINT := 21;
	INDEX_GIVENRUNNINGCOMMAND_WHENPAUSE_EXPECTCOMMANDTRANSITIONSTOPAUSEDSTATE		: DINT := 22;
	INDEX_GIVENTIMERSTARTED_WHENCYCLICLOGICRUNS_EXPECTELAPSEDTIMEINCREASES			: DINT := 23;
	INDEX_GIVENTIMERSTOPPED_WHENCYCLICLOGICRUNS_EXPECTELAPSEDTIMEREMAINCONSTANT		: DINT := 24;
	INDEX_GIVENVALIDCONFIGURATION_WHENINJECTCONFIGURATIONCALLED_EXPECTCONFIGSTORED	: DINT := 25;

	// TEST_* methods (26-113)
	INDEX_ABORT_AFTERCOMPLETE_IGNOREDWITHWARNING									: DINT := 26;
	INDEX_ABORT_ERRORCLASSIFICATION													: DINT := 27;
	INDEX_ABORT_WHENIDLEQUEUED_SETSRESULTABORTED									: DINT := 28;
	INDEX_ABORTAFTERCOMPLETE_STATEPRESERVATION										: DINT := 29;
	INDEX_ABORTDURINGCOMPLETIONWAIT													: DINT := 30;
	INDEX_ACCEPTEDCOMMAND_WHENEXECUTED_RESULTBECOMESOK								: DINT := 31;
	INDEX_BADREQUEST_INTERLOCKMISCONFIGURED											: DINT := 32;
	INDEX_BUSYCOMMANDELAPSEDTIMEEQUALS_COMMANDABORTED								: DINT := 33;
	INDEX_CANCEL_FROMQUEUEDSTATE													: DINT := 34;
	INDEX_CANCEL_REMOVESCOMMANDFROMQUEUE											: DINT := 35;
	INDEX_CANCEL_SETSCOMMANDSTATUSTOCANCELLED										: DINT := 36;
	INDEX_CANCEL_SETSRESULTCANCELLED												: DINT := 37;
	INDEX_CANCEL_WHENBUSY_REJECTED_NOCHANGETOSTATE									: DINT := 38;
	INDEX_COMMAND_LOCALREFERENCES_INITIALIZEDPROPERLY								: DINT := 39;
	INDEX_COMMAND_MISSINGCONFIGINTERFACE_FALLBACK									: DINT := 40;
	INDEX_COMMAND_PERMINTLKCHILD_INITIALIZED										: DINT := 41;
	INDEX_COMMANDATTEMPTSEXCEEDRETRYCOUNT											: DINT := 42;
	INDEX_COMMANDCOMPLETES_STATUSDONEANDCLEARED										: DINT := 43;
	INDEX_COMMANDSTATUS_CONFIGREF_POINTSTOCONFIGURATION								: DINT := 44;
	INDEX_COMMANDTIMEOUT_TRIGGERSRESET												: DINT := 45;
	INDEX_COMPLETE_ERROR_PERSISTSUNTILRESET											: DINT := 46;
	INDEX_COMPLETE_OK_AUTORESETNEXTCYCLE											: DINT := 47;
	INDEX_COMPLETESTATE_PRESERVESABORTEDRESULT										: DINT := 48;
	INDEX_COMPLETESTATE_PRESERVESTIMEOUTRESULT										: DINT := 49;
	INDEX_COMPLETESTATE_SETSOKFORSUCCESSFUL											: DINT := 50;
	INDEX_COMPLETIONCALLBACKTOSEQUENCER												: DINT := 51;
	INDEX_COMPLETIONCONDITIONEVALUATION												: DINT := 52;
	INDEX_COMPLETIONCONDITIONWITHTIMEOUT											: DINT := 53;
	INDEX_COMPLETIONWITHINTERLOCKDROP												: DINT := 54;
	INDEX_COMPLEXCOMPLETIONCONDITION												: DINT := 55;
	INDEX_COMPONENTBUSY_DURINGVALIDATION_RESULTCONFLICT								: DINT := 56;
	INDEX_CONFIG_FALLBACKTOLOCAL_WHENINJECTEDINVALID								: DINT := 57;
	INDEX_CONFIG_RECOVERYTOINJECTED_WHENVALIDAGAIN									: DINT := 58;
	INDEX_CONFIGURATIONRESOLUTION_HANDLESVALIDINVALID								: DINT := 59;
	INDEX_CYCLICLOGIC_STATEMACHINEPROGRESSION										: DINT := 60;
	INDEX_DISCRETECOMPLETIONCONDITION												: DINT := 61;
	INDEX_DYNAMICCOMPLETIONCONDITIONUPDATE											: DINT := 62;
	INDEX_EDGETRIGGERED_STATEMACHINEEXECUTION										: DINT := 63;
	INDEX_EXECUTE_HAPPYPATH_TRANSITIONSTOMONITOR									: DINT := 64;
	INDEX_EXECUTE_STATEMACHINEPROGRESSION											: DINT := 65;
	INDEX_EXECUTE_TRANSITIONSFROMACCEPTEDTOOK										: DINT := 66;
	INDEX_EXECUTE_VALIDATESBEFOREACCEPTING											: DINT := 67;
	INDEX_EXECUTE_WHENPERMISSIVEMISSING_RETURNSFORBIDDEN							: DINT := 68;
	INDEX_FASTCOMPLETIONINONESCAN													: DINT := 69;
	INDEX_FORBIDDEN_RESUMEWITHOUTPERMISSIVE											: DINT := 70;
	INDEX_INJECTCONFIGURATIONS_STORESINTERFACES										: DINT := 71;
	INDEX_INTERFACEINJECTIONCONFIGURATIONRESOLUTION									: DINT := 72;
	INDEX_INTERLOCKDROP_ABORTSCOMMANDWHENCONFIGURED									: DINT := 73;
	INDEX_INTERLOCKDROP_FROMMONITORSTATE											: DINT := 74;
	INDEX_INTERLOCKINVALIDCONFIG_DURINGVALIDATION									: DINT := 75;
	INDEX_INTERLOCKLOST_COMPREHENSIVESTATETRANSITIONS								: DINT := 76;
	INDEX_INTERLOCKLOST_FROMEXECUTESTATE											: DINT := 77;
	INDEX_INTERLOCKLOST_SETSCORRECTRESULT											: DINT := 78;
	INDEX_INTERLOCKREFERENCELOST_DURINGEXECUTION									: DINT := 79;
	INDEX_METHODENABLEMENT_BUSYSTATE_ALLOWABORT										: DINT := 80;
	INDEX_METHODENABLEMENT_DONESTATE_ALLOWRESET										: DINT := 81;
	INDEX_METHODENABLEMENT_IDLEWITHINTERLOK_ALLOWEXECUTE							: DINT := 82;
	INDEX_METHODENABLEMENT_IDLEWITHOUTINTERLOK_REJECT								: DINT := 83;
	INDEX_MOTIONCOMPLETIONCONDITION													: DINT := 84;
	INDEX_OPERATIONTOCOMMANDTRANSLATION												: DINT := 85;
	INDEX_OPERATORABORT_VSINTERLOCKABORT_DIFFERENTRESULTS							: DINT := 86;
	INDEX_PAUSERESUME_STATETRANSITIONS												: DINT := 87;
	INDEX_PAUSERESUMEWITHCOMPLETIONCONDITION										: DINT := 88;
	INDEX_PERMINTLKLOST_DURINGBUSY_COMMANDABORTED									: DINT := 89;
	INDEX_PERMISSIVEFALSE_DURINGVALIDATION_FORBIDDEN								: DINT := 90;
	INDEX_QUEUEOPERATIONS_MULTIPLECOMMANDSATOMICITY									: DINT := 91;
	INDEX_RECIPEMANAGERPROVIDESCOMMANDCONFIG										: DINT := 92;
	INDEX_RESET_CLEARSCOMMANDSTATE													: DINT := 93;
	INDEX_RESULTPERSISTENCE_TERMINALSTATES											: DINT := 94;
	INDEX_RETRYCOUNT_INCREMENTONEXECUTIONSTARTONLY									: DINT := 95;
	INDEX_RUNTIMECOMMANDCONFIGLOSS_INJECTEDREFSINVALIDATED							: DINT := 96;
	INDEX_RUNTIMECOMMANDCONFIGRECOVERY_VALIDREFSRESTORED							: DINT := 97;
	INDEX_SLOWCOMPLETIONMULTIPLESCANS												: DINT := 98;
	INDEX_STEPSTATE_TRANSITIONSANDVALIDATION										: DINT := 99;
	INDEX_SYSTEMATICSTATEVALIDATION_IDLESTATES										: DINT := 100;
	INDEX_SYSTEMATICSTATEVALIDATION_TERMINALSTATES									: DINT := 101;
	INDEX_TERMINALRESULTS_ERRORFLAGCONSISTENCY										: DINT := 102;
	INDEX_TIMEBASEDCOMPLETIONCONDITION												: DINT := 103;
	INDEX_TIMEOUTANDINTERLOCKLOST_SAMECYCLE_PRIORITIZE								: DINT := 104;
	INDEX_TIMERCOMPLETIONTIME_SETONCOMMANDCOMPLETE									: DINT := 105;
	INDEX_TIMERINTEGRATION_WITHCOMMANDSTATEMACHINE									: DINT := 106;
	INDEX_TIMERPAUSERESUME_ELAPSEDTIMEACCURACY										: DINT := 107;
	INDEX_TIMERSTOPSONCOMMANDCOMPLETE_NOTTIMEOUT									: DINT := 108;
	INDEX_TIMERTRIGGERTIME_SETONCOMMANDSTART										: DINT := 109;
	INDEX_VALIDATE_RETURNSPROPERRESULT												: DINT := 110;
	INDEX_VALIDATE_WITHCONTINUOUSEVALUATION											: DINT := 111;
	INDEX_VALIDATIONOK_INTERLOCKDROP_DURINGEXECUTION								: DINT := 112;
	INDEX_VALIDCOMMAND_EXPECTEXECUTED												: DINT := 113;

	// Additional indices for multi-scenario tests
	INDEX_TERMINALRESULTS_CLEANCANCEL												: DINT := 114;
	INDEX_TERMINALRESULTS_INTERLOCKLOST											: DINT := 115;
	INDEX_TERMINALRESULTS_TIMEOUT													: DINT := 116;
	INDEX_TERMINALRESULTS_COMPLETE_OK												: DINT := 117;
	INDEX_TERMINALRESULTS_COMPLETE_ERROR											: DINT := 118;
	INDEX_VALIDATIONOK_INTERLOCKDROP_SCENARIO2										: DINT := 119;

	// Fixed duplicate indices - these tests were incorrectly reusing other test indices
	INDEX_TIMEOUTANDINTERLOCKLOST_SAMECYCLE_PRIORITIZEINTERLOCKLOST					: DINT := 120;
	INDEX_VALIDATE_RETURNSPROPERRESULTBASEDONPERMISSIVES							: DINT := 121;
	INDEX_VALIDATE_WITHCONTINUOUSEVALUATION_PROPER									: DINT := 122;
	INDEX_VALIDATIONOK_INTERLOCKDROPDURINGEXECUTION									: DINT := 123;
	INDEX_VALIDCOMMAND_EXPECTEXECUTED_PROPER										: DINT := 124;
END_VAR

VAR

	// Mock component for testing
	MockComponent 			: FB_ComponentDerivative;

	// Common test interfaces for all methods (FB-level for stability)
	// Initialized to 0 to prevent page faults - will be set by each test method safely
	iTestCommand 			: I_CommandUnderTest;
	iTestCommandConfig 		: I_CommandConfiguration;
	iTestComponent 			: I_ComponentFull;
	iTestPermIntlkConfig 	: I_PermIntlkConfiguration;
	iTestPermIntlk 			: I_PermIntlk;
	iTestPermIntlkEval		: I_PermIntlk;
	
	// Array instances for test methods (indices 0-17)
	TestCommand : ARRAY[GC_Test.INDEX_TestFB_Command_MIN..GC_Test.INDEX_TestFB_Command_MAX] OF FB_CommandUnderTest;
	TestComponent : ARRAY[GC_Test.INDEX_TestFB_Command_MIN..GC_Test.INDEX_TestFB_Command_MAX] OF FB_ComponentDerivative;
	TestCommandConfig : ARRAY[GC_Test.INDEX_TestFB_Command_MIN..GC_Test.INDEX_TestFB_Command_MAX] OF FB_CmdPermIntlkConfiguration;
	TestPermIntlk : ARRAY[GC_Test.INDEX_TestFB_Command_MIN..GC_Test.INDEX_TestFB_Command_MAX] OF FB_PermIntlkCommand;
	MockQueue : ARRAY[GC_Test.INDEX_TestFB_Command_MIN..GC_Test.INDEX_TestFB_Command_MAX] OF FB_RingBufferICmd;
	CommandTimer : ARRAY[GC_Test.INDEX_TestFB_Command_MIN..GC_Test.INDEX_TestFB_Command_MAX] OF FB_CommandElapsedTimer;
//	FileHandler : ARRAY[GC_Test.INDEX_TestFB_Command_MIN..GC_Test.INDEX_TestFB_Command_MAX] OF FB_FileHandlerCsv;
END_VAR

// === Missing Timer Tests ===
TEST_TimerCompletionTime_SetOnCommandComplete();
TEST_TimerIntegration_WithCommandStateMachine(); //stack overflow?
TEST_TimerPauseResume_ElapsedTimeAccuracy(); //stack overflow?
TEST_TimerStopsOnCommandComplete_NotTimeout();
TEST_TimerTriggerTime_SetOnCommandStart();

// === Missing Interlock Tests ===
TEST_InterlockDrop_AbortsCommandWhenConfigured();
TEST_InterlockDrop_FromMonitorState_CommandAborted();
TEST_InterlockInvalidConfigurationDuringValidation_ReturnsBadRequest();
TEST_InterlockLost_ComprehensiveStateTransitions();
TEST_InterlockLost_FromExecuteState();
TEST_InterlockLost_SetsCorrectResult();
TEST_InterlockReferenceLostDuringExecution_FallsBackOrAborts();

// === Missing Method Enablement Tests ===
TEST_MethodEnablement_BusyState_ShouldAllowAbortRejectExecute();
TEST_MethodEnablement_DoneState_ShouldAllowResetRejectExecute();
TEST_MethodEnablement_IdleWithInterlockOK_ShouldAllowExecute();
TEST_MethodEnablement_IdleWithoutInterlockOK_ShouldRejectExecute();

METHOD PRIVATE TEST_MethodEnablement_BusyState_ShouldAllowAbortRejectExecute
VAR
	TestIdx : DINT := INDEX_METHODENABLEMENT_BUSYSTATE_ALLOWABORT;
    stCommandStatus : ST_CommandStatus;
	stBaseStatus	: ST_BaseStatus;
    eAbortResult : E_CommandResult;
    eExecuteResult : E_CommandResult;
END_VAR
TEST(__POUNAME());

// REAL TEST: InputMask 1 (Busy=1) should enable Abort, disable Execute
// From CSV: EnabledMethods="Pause" (Abort available via expression, Execute NOT enabled)

// Initialize test objects
TestCommand[TestIdx].Initialize();
TestComponent[TestIdx].Initialize();
TestCommandConfig[TestIdx].Initialize();

stCommandStatus.BaseStatus REF= stBaseStatus;

// Safe interface assignments  
iTestCommand := TestCommand[TestIdx];

iTestCommandConfig := TestCommandConfig[TestIdx];

iTestComponent := TestComponent[TestIdx];

IF iTestCommandConfig <> 0 THEN
	stCommandStatus.ConfigRef REF= iTestCommandConfig.P_CommandConfiguration;
END_IF

// Configure command
iTestCommandConfig.P_CommandConfiguration.CommandDescription := 'Method Enablement Test - Busy State Methods';

// Setup command with configurations
iTestCommand.InjectConfigurations(
    iComponent := iTestComponent,
    iCommandConfiguration := iTestCommandConfig,
    iPermIntlkConfiguration := iTestPermIntlkConfig
);

// Create InputMask 1 state: Busy=TRUE, all others FALSE
stCommandStatus.BaseStatus.Busy := TRUE;   // Bit 0 = InputMask 1
stCommandStatus.BaseStatus.Error := FALSE;
stCommandStatus.BaseStatus.Done := FALSE;
stCommandStatus.ConfigRef.PermIntlkConfiguredAsInterlock := FALSE;
stCommandStatus.ConfigRef.AbortOnInterlockDrop := FALSE;
// TRUE := FALSE;
// FALSE := FALSE;

// Inject busy state
iTestCommand.SetCommandStatus(stCommandStatus);

// REAL TEST 1: Try Abort() - should succeed in busy state
iTestCommand.Abort();

// Verify Abort was accepted by checking command status
AssertEquals_UDINT(
    Expected := E_CommandResult.Aborted,
    Actual := iTestCommand.P_CommandStatus.Result,
    Message := 'Abort should be accepted in busy state (InputMask 1)'
);

// Reset to busy state for second test
iTestCommand.SetCommandStatus(stCommandStatus);

// REAL TEST 2: Try Execute() - should fail in busy state (conflict)
iTestCommand.Execute();

// Verify Execute was rejected due to conflict
AssertEquals_UDINT(
    Expected := E_CommandResult.Forbidden,
    Actual := iTestCommand.P_CommandStatus.Result,
    Message := 'Execute should be rejected with Conflict in busy state (InputMask 1)'
);

TEST_FINISHED();
END_METHOD

METHOD PRIVATE TEST_MethodEnablement_DoneState_ShouldAllowResetRejectExecute
VAR
	TestIdx : DINT := INDEX_METHODENABLEMENT_DONESTATE_ALLOWRESET;
    stCommandStatus : ST_CommandStatus;
	stBaseStatus	: ST_BaseStatus;
    eResetResult : E_CommandResult;
    eExecuteResult : E_CommandResult;
END_VAR
TEST(__POUNAME());

// REAL TEST: InputMask 4 (Done=1) should enable Reset, disable Execute  
// From CSV: EnabledMethods="Queue,Reset" (Reset available, Execute NOT enabled)

// Initialize test objects
TestCommand[TestIdx].Initialize();
TestComponent[TestIdx].Initialize();
TestCommandConfig[TestIdx].Initialize();

stCommandStatus.BaseStatus REF= stBaseStatus;

